  MoveL (T18849) to (113.75, 117.08, 19.7) mm, rotated rx 180 ry 0 rz -180 deg; joints [1.869, 69.168, -34.061, 3.247, -35.151, -2.656]
  Call Extruder 0.34538
  MoveL (T18850) to (108.6, 106.98, 19.7) mm, rotated rx 180 ry 0 rz -180 deg; joints [1.874, 68.733, -33.242, 3.226, -35.533, -2.626]
  Call Extruder 0.01947
  MoveL (T18851) to (108.6, 106.34, 19.7) mm, rotated rx 180 ry 0 rz -180 deg; joints [1.874, 68.733, -33.242, 3.226, -35.533, -2.626]
  Set speed (150.0 mm/s)
  MoveL (T18852) to (108.54, 105.89, 19.7) mm, rotated rx 180 ry 0 rz -180 deg; joints [1.874, 68.733, -33.242, 3.226, -35.533, -2.626]
  Set speed (45.0 mm/s)
  Call Extruder -1.6
  MoveL (T18853) to (108.54, 105.89, 19.7) mm, rotated rx 180 ry 0 rz -180 deg; joints [1.866, 68.675, -33.134, 3.208, -35.583, -2.61]
  Set speed (120.0 mm/s)
  MoveL (T18854) to (108.54, 105.89, 19.7) mm, rotated rx 180 ry 0 rz -180 deg; joints [1.866, 68.675, -33.134, 3.208, -35.583, -2.61]
  Call Extruder -0.38
  MoveL (T18855) to (109.66, 106.33, 19.7) mm, rotated rx 180 ry 0 rz -180 deg; joints [1.815, 68.53, -32.862, 3.11, -35.708, -2.526]
  Set speed (45.0 mm/s)
  Call Extruder -0.02
  MoveL (T18856) to (109.66, 106.33, 19.7) mm, rotated rx 180 ry 0 rz -180 deg; joints [1.815, 68.53, -32.862, 3.11, -35.708, -2.526]
  Set speed (150.0 mm/s)
  MoveL (T18857) to (109.66, 106.33, 21.7) mm, rotated rx 180 ry 0 rz -180 deg; joints [2.818, 66.213, -28.512, 4.602, -37.791, -3.64]
  MoveL (T18858) to (104.34, 103.54, 21.7) mm, rotated rx 180 ry 0 rz -180 deg; joints [2.818, 66.213, -28.512, 4.602, -37.791, -3.64]
  MoveL (T18859) to (104.34, 103.54, 19.7) mm, rotated rx 180 ry 0 rz -180 deg; joints [2.938, 66.228, -28.539, 4.799, -37.786, -3.796]
  Set speed (40.0 mm/s)
  Call Extruder 2.0
  MoveL (T18860) to (104.34, 103.54, 19.7) mm, rotated rx 180 ry 0 rz -180 deg; joints [2.938, 66.228, -28.539, 4.799, -37.786, -3.796]
  Call Extruder 0.52159
  MoveL (T18861) to (121.46, 103.54, 19.7) mm, rotated rx 180 ry 0 rz -180 deg; joints [2.938, 66.228, -28.539, 4.799, -37.786, -3.796]
  Call Extruder 0.54596
  MoveL (T18862) to (121.46, 121.46, 19.7) mm, rotated rx 180 ry 0 rz -180 deg; joints [2.938, 66.228, -28.539, 4.799, -37.786, -3.796]
  Call Extruder 0.54596
  MoveL (T18863) to (103.54, 121.46, 19.7) mm, rotated rx 180 ry 0 rz -180 deg; joints [3.295, 67.194, -30.352, 5.484, -36.967, -4.386]
  Call Extruder 0.54596
  MoveL (T18864) to (103.54, 103.54, 19.7) mm, rotated rx 180 ry 0 rz -180 deg; joints [3.288, 67.492, -30.912, 5.506, -36.706, -4.419]
  Call Extruder 0.02254
  MoveL (T18865) to (104.28, 103.54, 19.7) mm, rotated rx 180 ry 0 rz -180 deg; joints [3.288, 67.492, -30.912, 5.506, -36.706, -4.419]
  Set speed (150.0 mm/s)
  MoveL (T18866) to (103.53, 103.13, 19.7) mm, rotated rx 180 ry 0 rz -180 deg; joints [3.288, 67.492, -30.912, 5.506, -36.706, -4.419]
  Set speed (40.0 mm/s)
  MoveL (T18867) to (103.53, 103.13, 19.7) mm, rotated rx 180 ry 0 rz -180 deg; joints [2.356, 69.73, -35.116, 4.142, -34.684, -3.408]
  Call Extruder 0.55858
  MoveL (T18868) to (121.87, 103.13, 19.7) mm, rotated rx 180 ry 0 rz -180 deg; joints [2.356, 69.73, -35.116, 4.142, -34.684, -3.408]
  Call Extruder 0.57077
  MoveL (T18869) to (121.87, 121.87, 19.7) mm, rotated rx 180 ry 0 rz -180 deg; joints [2.29, 69.723, -35.102, 4.026, -34.687, -3.312]
  Call Extruder 0.57077
  MoveL (T18870) to (103.13, 121.87, 19.7) mm, rotated rx 180 ry 0 rz -180 deg; joints [2.29, 69.723, -35.102, 4.026, -34.687, -3.312]
  Call Extruder 0.57077
  MoveL (T18871) to (103.13, 103.13, 19.7) mm, rotated rx 180 ry 0 rz -180 deg; joints [1.775, 68.231, -32.301, 3.023, -35.968, -2.447]
  Call Extruder 0.01036
  MoveL (T18872) to (103.47, 103.13, 19.7) mm, rotated rx 180 ry 0 rz -180 deg; joints [1.775, 68.231, -32.301, 3.023, -35.968, -2.447]
  Set speed (150.0 mm/s)
  MoveL (T18873) to (102.72, 102.81, 19.7) mm, rotated rx 180 ry 0 rz -180 deg; joints [1.875, 67.989, -31.846, 3.176, -36.185, -2.565]
  Set speed (25.0 mm/s)
  MoveL (T18874) to (102.72, 102.81, 19.7) mm, rotated rx 180 ry 0 rz -180 deg; joints [1.875, 67.989, -31.846, 3.176, -36.185, -2.565]
  Call Extruder 0.00259
  MoveL (T18875) to (102.72, 102.72, 19.7) mm, rotated rx 180 ry 0 rz -180 deg; joints [1.875, 67.989, -31.846, 3.176, -36.185, -2.565]
  Call Extruder 0.59557
  MoveL (T18876) to (122.28, 102.72, 19.7) mm, rotated rx 180 ry 0 rz -180 deg; joints [1.875, 67.989, -31.846, 3.176, -36.185, -2.565]
  Call Extruder 0.59557
  MoveL (T18877) to (122.28, 122.28, 19.7) mm, rotated rx 180 ry 0 rz -180 deg; joints [1.884, 67.935, -31.744, 3.189, -36.233, -2.573]
  Call Extruder 0.59557
  MoveL (T18878) to (102.72, 122.28, 19.7) mm, rotated rx 180 ry 0 rz -180 deg; joints [1.888, 67.676, -31.258, 3.177, -36.46, -2.556]
  Call Extruder 0.59115
  MoveL (T18879) to (102.72, 102.87, 19.7) mm, rotated rx 180 ry 0 rz -180 deg; joints [1.888, 67.676, -31.258, 3.177, -36.46, -2.556]
  Set speed (150.0 mm/s)
  MoveL (T18880) to (102.78, 102.75, 19.7) mm, rotated rx 180 ry 0 rz -180 deg; joints [1.888, 67.676, -31.258, 3.177, -36.46, -2.556]
  Set speed (45.0 mm/s)
  Call Extruder -1.6
  MoveL (T18881) to (102.78, 102.75, 19.7) mm, rotated rx 180 ry 0 rz -180 deg; joints [1.888, 67.676, -31.258, 3.177, -36.46, -2.556]
  Set speed (120.0 mm/s)
  MoveL (T18882) to (102.78, 102.75, 19.7) mm, rotated rx 180 ry 0 rz -180 deg; joints [1.888, 67.676, -31.258, 3.177, -36.46, -2.556]
  Call Extruder -0.05166
  MoveL (T18883) to (102.72, 102.72, 19.7) mm, rotated rx 180 ry 0 rz -180 deg; joints [1.888, 67.676, -31.258, 3.177, -36.46, -2.556]
  Call Extruder -0.32834
  MoveL (T18884) to (103.65, 102.72, 19.7) mm, rotated rx 180 ry 0 rz -180 deg; joints [1.888, 67.676, -31.258, 3.177, -36.46, -2.556]
  Set speed (45.0 mm/s)
  Call Extruder -0.02
  MoveL (T18885) to (103.65, 102.72, 19.7) mm, rotated rx 180 ry 0 rz -180 deg; joints [1.888, 67.676, -31.258, 3.177, -36.46, -2.556]
  Set speed (150.0 mm/s)
  MoveL (T18886) to (103.65, 102.72, 21.7) mm, rotated rx 180 ry 0 rz -180 deg; joints [1.888, 67.676, -31.258, 3.177, -36.46, -2.556]
  MoveL (T18887) to (121.34, 120.51, 21.7) mm, rotated rx 180 ry 0 rz -180 deg; joints [1.884, 67.935, -31.744, 3.189, -36.233, -2.573]
  MoveL (T18888) to (121.34, 120.51, 19.7) mm, rotated rx 180 ry 0 rz -180 deg; joints [1.884, 67.935, -31.744, 3.189, -36.233, -2.573]
  Set speed (40.0 mm/s)
  Call Extruder 2.0
  MoveL (T18889) to (121.34, 120.51, 19.7) mm, rotated rx 180 ry 0 rz -180 deg; joints [1.884, 67.935, -31.744, 3.189, -36.233, -2.573]
  Call Extruder 0.02815
  MoveL (T18890) to (120.69, 121.16, 19.7) mm, rotated rx 180 ry 0 rz -180 deg; joints [1.879, 67.965, -31.801, 3.182, -36.206, -2.568]
  Call Extruder 0.01786
  MoveL (T18891) to (120.11, 121.16, 19.7) mm, rotated rx 180 ry 0 rz -180 deg; joints [1.879, 67.965, -31.801, 3.182, -36.206, -2.568]
  Call Extruder 0.04544
  MoveL (T18892) to (121.16, 120.11, 19.7) mm, rotated rx 180 ry 0 rz -180 deg; joints [1.879, 67.965, -31.801, 3.182, -36.206, -2.568]
  Call Extruder 0.01786
  MoveL (T18893) to (121.16, 119.53, 19.7) mm, rotated rx 180 ry 0 rz -180 deg; joints [1.879, 67.965, -31.801, 3.182, -36.206, -2.568]
  Call Extruder 0.0707
  MoveL (T18894) to (119.53, 121.16, 19.7) mm, rotated rx 180 ry 0 rz -180 deg; joints [1.879, 67.965, -31.801, 3.182, -36.206, -2.568]
  Call Extruder 0.01786
  MoveL (T18895) to (118.95, 121.16, 19.7) mm, rotated rx 180 ry 0 rz -180 deg; joints [1.879, 67.731, -31.763, 3.197, -36.01, -2.587]
  Call Extruder 0.09595
  MoveL (T18896) to (121.16, 118.95, 19.7) mm, rotated rx 180 ry 0 rz -180 deg; joints [1.476, 70.466, -36.894, 2.667, -33.601, -2.222]
  Call Extruder 0.01786
  MoveL (T18897) to (121.16, 118.37, 19.7) mm, rotated rx 180 ry 0 rz -180 deg; joints [1.476, 70.698, -36.935, 2.654, -33.792, -2.206]
  Call Extruder 0.12121
  MoveL (T18898) to (118.37, 121.16, 19.7) mm, rotated rx 180 ry 0 rz -180 deg; joints [1.476, 70.698, -36.935, 2.654, -33.792, -2.206]
  Call Extruder 0.01786
  MoveL (T18899) to (117.79, 121.16, 19.7) mm, rotated rx 180 ry 0 rz -180 deg; joints [1.476, 70.698, -36.935, 2.654, -33.792, -2.206]
  Call Extruder 0.14646
  MoveL (T18900) to (121.16, 117.79, 19.7) mm, rotated rx 180 ry 0 rz -180 deg; joints [1.476, 70.698, -36.935, 2.654, -33.792, -2.206]
  Call Extruder 0.01786
  MoveL (T18901) to (121.16, 117.21, 19.7) mm, rotated rx 180 ry 0 rz -180 deg; joints [1.476, 70.698, -36.935, 2.654, -33.792, -2.206]
  Call Extruder 0.17172
  MoveL (T18902) to (117.21, 121.16, 19.7) mm, rotated rx 180 ry 0 rz -180 deg; joints [1.476, 70.698, -36.935, 2.654, -33.792, -2.206]
  Call Extruder 0.01786
  MoveL (T18903) to (116.62, 121.16, 19.7) mm, rotated rx 180 ry 0 rz -180 deg; joints [1.476, 70.698, -36.935, 2.654, -33.792, -2.206]
  Call Extruder 0.19697
  MoveL (T18904) to (121.16, 116.62, 19.7) mm, rotated rx 180 ry 0 rz -180 deg; joints [1.476, 70.698, -36.935, 2.654, -33.792, -2.206]
  Call Extruder 0.01786
  MoveL (T18905) to (121.16, 116.04, 19.7) mm, rotated rx 180 ry 0 rz -180 deg; joints [1.4, 70.466, -36.499, 2.505, -33.993, -2.077]
  Call Extruder 0.1471
  MoveL (T18906) to (117.77, 119.43, 19.7) mm, rotated rx 180 ry 0 rz -180 deg; joints [1.402, 70.285, -36.159, 2.497, -34.152, -2.067]
  Call Extruder 0.01786
  MoveL (T18907) to (117.77, 118.85, 19.7) mm, rotated rx 180 ry 0 rz -180 deg; joints [1.402, 70.285, -36.159, 2.497, -34.152, -2.067]
  Call Extruder 0.1471
  MoveL (T18908) to (121.16, 115.46, 19.7) mm, rotated rx 180 ry 0 rz -180 deg; joints [1.402, 70.285, -36.159, 2.497, -34.152, -2.067]
  Call Extruder 0.01786
  MoveL (T18909) to (121.16, 114.88, 19.7) mm, rotated rx 180 ry 0 rz -180 deg; joints [1.402, 70.285, -36.159, 2.497, -34.152, -2.067]
  Call Extruder 0.1471
  MoveL (T18910) to (117.77, 118.27, 19.7) mm, rotated rx 180 ry 0 rz -180 deg; joints [1.52, 70.645, -36.835, 2.729, -33.84, -2.268]
  Call Extruder 0.0059
  MoveL (T18911) to (117.77, 118.07, 19.7) mm, rotated rx 180 ry 0 rz -180 deg; joints [1.582, 70.65, -36.844, 2.842, -33.839, -2.361]
  Call Extruder 0.00889
  MoveL (T18912) to (117.64, 117.82, 19.7) mm, rotated rx 180 ry 0 rz -180 deg; joints [1.582, 70.65, -36.844, 2.842, -33.839, -2.361]
  Call Extruder 0.15283
  MoveL (T18913) to (121.16, 114.3, 19.7) mm, rotated rx 180 ry 0 rz -180 deg; joints [1.582, 70.65, -36.844, 2.842, -33.839, -2.361]
  Call Extruder 0.01786
  MoveL (T18914) to (121.16, 113.72, 19.7) mm, rotated rx 180 ry 0 rz -180 deg; joints [1.403, 70.106, -35.823, 2.49, -34.309, -2.057]
  Call Extruder 0.16138
  MoveL (T18915) to (117.44, 117.43, 19.7) mm, rotated rx 180 ry 0 rz -180 deg; joints [1.403, 70.106, -35.823, 2.49, -34.309, -2.057]
  Call Extruder 0.01327
  MoveL (T18916) to (117.25, 117.05, 19.7) mm, rotated rx 180 ry 0 rz -180 deg; joints [1.403, 70.106, -35.823, 2.49, -34.309, -2.057]
  Call Extruder 0.16993
  MoveL (T18917) to (121.16, 113.14, 19.7) mm, rotated rx 180 ry 0 rz -180 deg; joints [1.405, 69.928, -35.489, 2.483, -34.465, -2.047]
  Call Extruder 0.01786
  MoveL (T18918) to (121.16, 112.56, 19.7) mm, rotated rx 180 ry 0 rz -180 deg; joints [1.405, 69.928, -35.489, 2.483, -34.465, -2.047]
  Call Extruder 0.17848
  MoveL (T18919) to (117.05, 116.66, 19.7) mm, rotated rx 180 ry 0 rz -180 deg; joints [1.405, 69.928, -35.489, 2.483, -34.465, -2.047]
  Call Extruder 0.01327
  MoveL (T18920) to (116.85, 116.28, 19.7) mm, rotated rx 180 ry 0 rz -180 deg; joints [1.405, 69.928, -35.489, 2.483, -34.465, -2.047]
  Call Extruder 0.18703
  MoveL (T18921) to (121.16, 111.98, 19.7) mm, rotated rx 180 ry 0 rz -180 deg; joints [1.656, 70.504, -36.569, 2.965, -33.97, -2.459]
  Call Extruder 0.01786
  MoveL (T18922) to (121.16, 111.4, 19.7) mm, rotated rx 180 ry 0 rz -180 deg; joints [1.656, 70.504, -36.569, 2.965, -33.97, -2.459]
  Call Extruder 0.19558
  MoveL (T18923) to (116.66, 115.89, 19.7) mm, rotated rx 180 ry 0 rz -180 deg; joints [1.406, 69.752, -35.158, 2.476, -34.62, -2.038]
  Call Extruder 0.01327
  MoveL (T18924) to (116.46, 115.51, 19.7) mm, rotated rx 180 ry 0 rz -180 deg; joints [1.406, 69.752, -35.158, 2.476, -34.62, -2.038]
  Call Extruder 0.20412
  MoveL (T18925) to (121.16, 110.81, 19.7) mm, rotated rx 180 ry 0 rz -180 deg; joints [1.408, 69.577, -34.828, 2.469, -34.773, -2.028]
  Call Extruder 0.01786
  MoveL (T18926) to (121.16, 110.23, 19.7) mm, rotated rx 180 ry 0 rz -180 deg; joints [1.408, 69.577, -34.828, 2.469, -34.773, -2.028]
  Call Extruder 0.21267
  MoveL (T18927) to (116.26, 115.13, 19.7) mm, rotated rx 180 ry 0 rz -180 deg; joints [1.688, 70.415, -36.404, 3.016, -34.049, -2.5]
  Call Extruder 0.01327
  MoveL (T18928) to (116.07, 114.74, 19.7) mm, rotated rx 180 ry 0 rz -180 deg; joints [1.688, 70.415, -36.404, 3.016, -34.049, -2.5]
  Call Extruder 0.22122
  MoveL (T18929) to (121.16, 109.65, 19.7) mm, rotated rx 180 ry 0 rz -180 deg; joints [1.688, 70.415, -36.404, 3.016, -34.049, -2.5]
  Call Extruder 0.01786
  MoveL (T18930) to (121.16, 109.07, 19.7) mm, rotated rx 180 ry 0 rz -180 deg; joints [1.72, 70.328, -36.239, 3.067, -34.127, -2.54]
  Call Extruder 0.22977
  MoveL (T18931) to (115.87, 114.36, 19.7) mm, rotated rx 180 ry 0 rz -180 deg; joints [1.72, 70.328, -36.239, 3.067, -34.127, -2.54]
  Call Extruder 0.01327
  MoveL (T18932) to (115.67, 113.97, 19.7) mm, rotated rx 180 ry 0 rz -180 deg; joints [1.72, 70.328, -36.239, 3.067, -34.127, -2.54]
  Call Extruder 0.23832
  MoveL (T18933) to (121.16, 108.49, 19.7) mm, rotated rx 180 ry 0 rz -180 deg; joints [1.409, 69.403, -34.502, 2.462, -34.926, -2.019]
  Call Extruder 0.01786
  MoveL (T18934) to (121.16, 107.91, 19.7) mm, rotated rx 180 ry 0 rz -180 deg; joints [1.409, 69.403, -34.502, 2.462, -34.926, -2.019]
  Call Extruder 0.24687
  MoveL (T18935) to (115.48, 113.59, 19.7) mm, rotated rx 180 ry 0 rz -180 deg; joints [1.411, 69.231, -34.178, 2.456, -35.077, -2.01]
  Call Extruder 0.01327
  MoveL (T18936) to (115.28, 113.2, 19.7) mm, rotated rx 180 ry 0 rz -180 deg; joints [1.411, 69.231, -34.178, 2.456, -35.077, -2.01]
  Call Extruder 0.25542
  MoveL (T18937) to (121.16, 107.33, 19.7) mm, rotated rx 180 ry 0 rz -180 deg; joints [1.411, 69.231, -34.178, 2.456, -35.077, -2.01]
  Call Extruder 0.01786
  MoveL (T18938) to (121.16, 106.75, 19.7) mm, rotated rx 180 ry 0 rz -180 deg; joints [1.753, 70.241, -36.076, 3.119, -34.205, -2.58]
  Call Extruder 0.26397
  MoveL (T18939) to (115.08, 112.82, 19.7) mm, rotated rx 180 ry 0 rz -180 deg; joints [1.753, 70.241, -36.076, 3.119, -34.205, -2.58]
  Call Extruder 0.01327
  MoveL (T18940) to (114.89, 112.44, 19.7) mm, rotated rx 180 ry 0 rz -180 deg; joints [1.753, 70.241, -36.076, 3.119, -34.205, -2.58]
  Call Extruder 0.27252
  MoveL (T18941) to (121.16, 106.17, 19.7) mm, rotated rx 180 ry 0 rz -180 deg; joints [1.785, 70.154, -35.913, 3.17, -34.282, -2.62]
  Call Extruder 0.01786
  MoveL (T18942) to (121.16, 105.59, 19.7) mm, rotated rx 180 ry 0 rz -180 deg; joints [1.785, 70.154, -35.913, 3.17, -34.282, -2.62]
  Call Extruder 0.13907
  MoveL (T18943) to (117.96, 108.79, 19.7) mm, rotated rx 180 ry 0 rz -180 deg; joints [1.785, 70.154, -35.913, 3.17, -34.282, -2.62]
  Call Extruder 0.01777
  MoveL (T18944) to (117.96, 109.36, 19.7) mm, rotated rx 180 ry 0 rz -180 deg; joints [1.412, 69.059, -33.856, 2.449, -35.228, -2.001]
  Call Extruder 0.01777
  MoveL (T18945) to (117.38, 109.36, 19.7) mm, rotated rx 180 ry 0 rz -180 deg; joints [1.412, 69.059, -33.856, 2.449, -35.228, -2.001]
  Call Extruder 0.11687
  MoveL (T18946) to (114.69, 112.05, 19.7) mm, rotated rx 180 ry 0 rz -180 deg; joints [1.414, 68.89, -33.537, 2.443, -35.377, -1.992]
  Call Extruder 0.01327
  MoveL (T18947) to (114.49, 111.67, 19.7) mm, rotated rx 180 ry 0 rz -180 deg; joints [1.414, 68.89, -33.537, 2.443, -35.377, -1.992]
  Call Extruder 0.10016
  MoveL (T18948) to (116.8, 109.36, 19.7) mm, rotated rx 180 ry 0 rz -180 deg; joints [1.815, 70.063, -35.741, 3.217, -34.364, -2.657]
  Call Extruder 0.01786
  MoveL (T18949) to (116.22, 109.36, 19.7) mm, rotated rx 180 ry 0 rz -180 deg; joints [1.815, 70.063, -35.741, 3.217, -34.364, -2.657]
  Call Extruder 0.08346
  MoveL (T18950) to (114.3, 111.28, 19.7) mm, rotated rx 180 ry 0 rz -180 deg; joints [1.817, 69.885, -35.407, 3.208, -34.52, -2.644]
  Call Extruder 0.01327
  MoveL (T18951) to (114.1, 110.9, 19.7) mm, rotated rx 180 ry 0 rz -180 deg; joints [1.817, 69.885, -35.407, 3.208, -34.52, -2.644]
  Call Extruder 0.06675
  MoveL (T18952) to (115.64, 109.36, 19.7) mm, rotated rx 180 ry 0 rz -180 deg; joints [1.416, 68.72, -33.22, 2.437, -35.525, -1.983]
  Call Extruder 0.01786
  MoveL (T18953) to (115.06, 109.36, 19.7) mm, rotated rx 180 ry 0 rz -180 deg; joints [1.416, 68.72, -33.22, 2.437, -35.525, -1.983]
  Call Extruder 0.05004
  MoveL (T18954) to (113.9, 110.52, 19.7) mm, rotated rx 180 ry 0 rz -180 deg; joints [1.416, 68.72, -33.22, 2.437, -35.525, -1.983]
  Call Extruder 0.01327
  MoveL (T18955) to (113.71, 110.13, 19.7) mm, rotated rx 180 ry 0 rz -180 deg; joints [1.417, 68.553, -32.905, 2.431, -35.672, -1.975]
  Call Extruder 0.03334
  MoveL (T18956) to (114.47, 109.36, 19.7) mm, rotated rx 180 ry 0 rz -180 deg; joints [1.417, 68.553, -32.905, 2.431, -35.672, -1.975]
  Call Extruder 0.01786
  MoveL (T18957) to (113.89, 109.36, 19.7) mm, rotated rx 180 ry 0 rz -180 deg; joints [1.417, 68.553, -32.905, 2.431, -35.672, -1.975]
  Call Extruder 0.02255
  MoveL (T18958) to (113.37, 109.88, 19.7) mm, rotated rx 180 ry 0 rz -180 deg; joints [1.819, 69.709, -35.077, 3.199, -34.674, -2.632]
  Set speed (45.0 mm/s)
  Call Extruder -1.6
  MoveL (T18959) to (113.37, 109.88, 19.7) mm, rotated rx 180 ry 0 rz -180 deg; joints [1.819, 69.709, -35.077, 3.199, -34.674, -2.632]
  Set speed (120.0 mm/s)
  MoveL (T18960) to (113.37, 109.88, 19.7) mm, rotated rx 180 ry 0 rz -180 deg; joints [1.819, 69.709, -35.077, 3.199, -34.674, -2.632]
  Call Extruder -0.26134
  MoveL (T18961) to (113.89, 109.36, 19.7) mm, rotated rx 180 ry 0 rz -180 deg; joints [1.821, 69.535, -34.749, 3.19, -34.827, -2.62]
  Call Extruder -0.11866
  MoveL (T18962) to (114.23, 109.36, 19.7) mm, rotated rx 180 ry 0 rz -180 deg; joints [1.821, 69.535, -34.749, 3.19, -34.827, -2.62]
  Set speed (45.0 mm/s)
  Call Extruder -0.02
  MoveL (T18963) to (114.23, 109.36, 19.7) mm, rotated rx 180 ry 0 rz -180 deg; joints [1.419, 68.386, -32.592, 2.425, -35.819, -1.966]
  Set speed (150.0 mm/s)
  MoveL (T18964) to (114.23, 109.36, 21.7) mm, rotated rx 180 ry 0 rz -180 deg; joints [1.419, 68.386, -32.592, 2.425, -35.819, -1.966]
  MoveL (T18965) to (117.77, 108.39, 21.7) mm, rotated rx 180 ry 0 rz -180 deg; joints [1.419, 68.386, -32.592, 2.425, -35.819, -1.966]
  MoveL (T18966) to (117.77, 108.39, 19.7) mm, rotated rx 180 ry 0 rz -180 deg; joints [1.42, 68.221, -32.281, 2.419, -35.964, -1.958]
  Set speed (40.0 mm/s)
  Call Extruder 2.0
  MoveL (T18967) to (117.77, 108.39, 19.7) mm, rotated rx 180 ry 0 rz -180 deg; joints [1.42, 68.221, -32.281, 2.419, -35.964, -1.958]
  Call Extruder 0.14703
  MoveL (T18968) to (121.16, 105.01, 19.7) mm, rotated rx 180 ry 0 rz -180 deg; joints [1.823, 69.361, -34.423, 3.182, -34.98, -2.608]
  Call Extruder 0.01786
  MoveL (T18969) to (121.16, 104.42, 19.7) mm, rotated rx 180 ry 0 rz -180 deg; joints [1.823, 69.361, -34.423, 3.182, -34.98, -2.608]
  Call Extruder 0.13907
  MoveL (T18970) to (117.96, 107.62, 19.7) mm, rotated rx 180 ry 0 rz -180 deg; joints [1.823, 69.361, -34.423, 3.182, -34.98, -2.608]
  Call Extruder 0.01786
  MoveL (T18971) to (117.96, 107.04, 19.7) mm, rotated rx 180 ry 0 rz -180 deg; joints [1.825, 69.189, -34.1, 3.173, -35.131, -2.596]
  Call Extruder 0.13906
  MoveL (T18972) to (121.16, 103.84, 19.7) mm, rotated rx 180 ry 0 rz -180 deg; joints [1.825, 69.189, -34.1, 3.173, -35.131, -2.596]
  Call Extruder 0.01786
  MoveL (T18973) to (120.58, 103.84, 19.7) mm, rotated rx 180 ry 0 rz -180 deg; joints [1.422, 68.056, -31.973, 2.413, -36.108, -1.95]
  Call Extruder 0.11381
  MoveL (T18974) to (117.96, 106.46, 19.7) mm, rotated rx 180 ry 0 rz -180 deg; joints [1.422, 68.056, -31.973, 2.413, -36.108, -1.95]
  Call Extruder 0.01786
  MoveL (T18975) to (117.96, 105.88, 19.7) mm, rotated rx 180 ry 0 rz -180 deg; joints [1.422, 68.056, -31.973, 2.413, -36.108, -1.95]
  Call Extruder 0.08856
  MoveL (T18976) to (119.99, 103.84, 19.7) mm, rotated rx 180 ry 0 rz -180 deg; joints [1.423, 67.893, -31.665, 2.408, -36.252, -1.942]
  Call Extruder 0.01786
  MoveL (T18977) to (119.41, 103.84, 19.7) mm, rotated rx 180 ry 0 rz -180 deg; joints [1.423, 67.893, -31.665, 2.408, -36.252, -1.942]
  Call Extruder 0.0633
  MoveL (T18978) to (117.96, 105.3, 19.7) mm, rotated rx 180 ry 0 rz -180 deg; joints [1.827, 69.018, -33.778, 3.165, -35.281, -2.585]
  Call Extruder 0.00424
  MoveL (T18979) to (117.96, 105.16, 19.7) mm, rotated rx 180 ry 0 rz -180 deg; joints [1.827, 69.018, -33.778, 3.165, -35.281, -2.585]
  Call Extruder 0.01362
  MoveL (T18980) to (117.51, 105.16, 19.7) mm, rotated rx 180 ry 0 rz -180 deg; joints [1.827, 69.018, -33.778, 3.165, -35.281, -2.585]
  Call Extruder 0.0573
  MoveL (T18981) to (118.83, 103.84, 19.7) mm, rotated rx 180 ry 0 rz -180 deg; joints [1.829, 68.848, -33.46, 3.157, -35.43, -2.573]
  Call Extruder 0.01786
  MoveL (T18982) to (118.25, 103.84, 19.7) mm, rotated rx 180 ry 0 rz -180 deg; joints [1.829, 68.848, -33.46, 3.157, -35.43, -2.573]
  Call Extruder 0.0573
  MoveL (T18983) to (116.93, 105.16, 19.7) mm, rotated rx 180 ry 0 rz -180 deg; joints [1.829, 68.848, -33.46, 3.157, -35.43, -2.573]
  Call Extruder 0.01786
  MoveL (T18984) to (116.35, 105.16, 19.7) mm, rotated rx 180 ry 0 rz -180 deg; joints [1.425, 67.731, -31.361, 2.402, -36.394, -1.934]
  Call Extruder 0.0573
  MoveL (T18985) to (117.67, 103.84, 19.7) mm, rotated rx 180 ry 0 rz -180 deg; joints [1.425, 67.731, -31.361, 2.402, -36.394, -1.934]
  Call Extruder 0.01786
  MoveL (T18986) to (117.09, 103.84, 19.7) mm, rotated rx 180 ry 0 rz -180 deg; joints [1.425, 67.731, -31.361, 2.402, -36.394, -1.934]
  Call Extruder 0.0573
  MoveL (T18987) to (115.77, 105.16, 19.7) mm, rotated rx 180 ry 0 rz -180 deg; joints [1.427, 67.569, -31.058, 2.397, -36.535, -1.926]
  Call Extruder 0.01786
  MoveL (T18988) to (115.19, 105.16, 19.7) mm, rotated rx 180 ry 0 rz -180 deg; joints [1.427, 67.569, -31.058, 2.397, -36.535, -1.926]
  Call Extruder 0.0573
  MoveL (T18989) to (116.51, 103.84, 19.7) mm, rotated rx 180 ry 0 rz -180 deg; joints [1.69, 68.284, -32.4, 2.882, -35.919, -2.335]
  Call Extruder 0.01786
  MoveL (T18990) to (115.93, 103.84, 19.7) mm, rotated rx 180 ry 0 rz -180 deg; joints [1.69, 68.284, -32.4, 2.882, -35.919, -2.335]
  Call Extruder 0.0573
  MoveL (T18991) to (114.61, 105.16, 19.7) mm, rotated rx 180 ry 0 rz -180 deg; joints [1.723, 68.204, -32.249, 2.932, -35.99, -2.373]
  Call Extruder 0.01786
  MoveL (T18992) to (114.03, 105.16, 19.7) mm, rotated rx 180 ry 0 rz -180 deg; joints [1.723, 68.204, -32.249, 2.932, -35.99, -2.373]
  Call Extruder 0.0573
  MoveL (T18993) to (115.35, 103.84, 19.7) mm, rotated rx 180 ry 0 rz -180 deg; joints [1.723, 68.204, -32.249, 2.932, -35.99, -2.373]
  Call Extruder 0.01786
  MoveL (T18994) to (114.77, 103.84, 19.7) mm, rotated rx 180 ry 0 rz -180 deg; joints [1.428, 67.409, -30.757, 2.391, -36.676, -1.918]
  Call Extruder 0.0573
  MoveL (T18995) to (113.45, 105.16, 19.7) mm, rotated rx 180 ry 0 rz -180 deg; joints [1.428, 67.409, -30.757, 2.391, -36.676, -1.918]
  Call Extruder 0.01786
  MoveL (T18996) to (112.87, 105.16, 19.7) mm, rotated rx 180 ry 0 rz -180 deg; joints [1.428, 67.409, -30.757, 2.391, -36.676, -1.918]
  Call Extruder 0.0573
  MoveL (T18997) to (114.18, 103.84, 19.7) mm, rotated rx 180 ry 0 rz -180 deg; joints [1.43, 67.249, -30.457, 2.386, -36.816, -1.911]
  Call Extruder 0.01786
  MoveL (T18998) to (113.6, 103.84, 19.7) mm, rotated rx 180 ry 0 rz -180 deg; joints [1.43, 67.249, -30.457, 2.386, -36.816, -1.911]
  Call Extruder 0.0573
  MoveL (T18999) to (112.28, 105.16, 19.7) mm, rotated rx 180 ry 0 rz -180 deg; joints [1.755, 68.124, -32.099, 2.983, -36.062, -2.412]
  Call Extruder 0.01786
  MoveL (T19000) to (111.7, 105.16, 19.7) mm, rotated rx 180 ry 0 rz -180 deg; joints [1.788, 68.044, -31.95, 3.033, -36.133, -2.451]
  Call Extruder 0.0573
  MoveL (T19001) to (113.02, 103.84, 19.7) mm, rotated rx 180 ry 0 rz -180 deg; joints [1.788, 68.044, -31.95, 3.033, -36.133, -2.451]
  Call Extruder 0.01786
  MoveL (T19002) to (112.44, 103.84, 19.7) mm, rotated rx 180 ry 0 rz -180 deg; joints [1.431, 67.091, -30.16, 2.381, -36.955, -1.903]
  Call Extruder 0.0573
  MoveL (T19003) to (111.12, 105.16, 19.7) mm, rotated rx 180 ry 0 rz -180 deg; joints [1.431, 67.091, -30.16, 2.381, -36.955, -1.903]
  Call Extruder 0.01786
  MoveL (T19004) to (110.54, 105.16, 19.7) mm, rotated rx 180 ry 0 rz -180 deg; joints [1.431, 67.091, -30.16, 2.381, -36.955, -1.903]
  Call Extruder 0.0573
  MoveL (T19005) to (111.86, 103.84, 19.7) mm, rotated rx 180 ry 0 rz -180 deg; joints [1.433, 66.934, -29.865, 2.376, -37.093, -1.896]
  Call Extruder 0.01786
  MoveL (T19006) to (111.28, 103.84, 19.7) mm, rotated rx 180 ry 0 rz -180 deg; joints [1.433, 66.934, -29.865, 2.376, -37.093, -1.896]
  Call Extruder 0.0573
  MoveL (T19007) to (109.96, 105.16, 19.7) mm, rotated rx 180 ry 0 rz -180 deg; joints [1.433, 66.934, -29.865, 2.376, -37.093, -1.896]
  Call Extruder 0.01786
  MoveL (T19008) to (109.38, 105.16, 19.7) mm, rotated rx 180 ry 0 rz -180 deg; joints [1.821, 67.965, -31.801, 3.084, -36.203, -2.489]
  Call Extruder 0.0573
  MoveL (T19009) to (110.7, 103.84, 19.7) mm, rotated rx 180 ry 0 rz -180 deg; joints [1.821, 67.965, -31.801, 3.084, -36.203, -2.489]
  Call Extruder 0.01786
  MoveL (T19010) to (110.12, 103.84, 19.7) mm, rotated rx 180 ry 0 rz -180 deg; joints [1.821, 67.965, -31.801, 3.084, -36.203, -2.489]
  Call Extruder 0.0573
  MoveL (T19011) to (108.8, 105.16, 19.7) mm, rotated rx 180 ry 0 rz -180 deg; joints [1.838, 67.923, -31.721, 3.111, -36.242, -2.51]
  Call Extruder 0.01786
  MoveL (T19012) to (108.22, 105.16, 19.7) mm, rotated rx 180 ry 0 rz -180 deg; joints [1.838, 67.923, -31.721, 3.111, -36.242, -2.51]
  Call Extruder 0.06527
  MoveL (T19013) to (109.72, 103.66, 19.7) mm, rotated rx 180 ry 0 rz -180 deg; joints [1.838, 67.923, -31.721, 3.111, -36.242, -2.51]
  Set speed (45.0 mm/s)
  Call Extruder -1.6
  MoveL (T19014) to (109.72, 103.66, 19.7) mm, rotated rx 180 ry 0 rz -180 deg; joints [1.841, 67.909, -31.695, 3.114, -36.254, -2.512]
  Set speed (120.0 mm/s)
  MoveL (T19015) to (109.72, 103.66, 19.7) mm, rotated rx 180 ry 0 rz -180 deg; joints [1.841, 67.909, -31.695, 3.114, -36.254, -2.512]
  Call Extruder -0.38
  MoveL (T19016) to (108.97, 104.42, 19.7) mm, rotated rx 180 ry 0 rz -180 deg; joints [1.842, 67.853, -31.591, 3.112, -36.302, -2.509]
  Set speed (45.0 mm/s)
  Call Extruder -0.02
  MoveL (T19017) to (108.97, 104.42, 19.7) mm, rotated rx 180 ry 0 rz -180 deg; joints [1.435, 66.777, -29.571, 2.371, -37.23, -1.889]
  Set speed (150.0 mm/s)
  MoveL (T19018) to (108.97, 104.42, 21.7) mm, rotated rx 180 ry 0 rz -180 deg; joints [1.435, 66.777, -29.571, 2.371, -37.23, -1.889]
  MoveL (T19019) to (111.87, 115.45, 21.7) mm, rotated rx 180 ry 0 rz -180 deg; joints [1.435, 66.777, -29.571, 2.371, -37.23, -1.889]
  MoveL (T19020) to (111.87, 115.45, 19.7) mm, rotated rx 180 ry 0 rz -180 deg; joints [1.435, 66.777, -29.571, 2.371, -37.23, -1.889]
  Set speed (40.0 mm/s)
  Call Extruder 2.0
  MoveL (T19021) to (111.87, 115.45, 19.7) mm, rotated rx 180 ry 0 rz -180 deg; joints [1.436, 66.621, -29.279, 2.367, -37.367, -1.881]
  Call Extruder 0.022
  MoveL (T19022) to (111.36, 115.96, 19.7) mm, rotated rx 180 ry 0 rz -180 deg; joints [1.436, 66.621, -29.279, 2.367, -37.367, -1.881]
  Call Extruder 0.01786
  MoveL (T19023) to (110.78, 115.96, 19.7) mm, rotated rx 180 ry 0 rz -180 deg; joints [1.844, 67.691, -31.287, 3.105, -36.444, -2.498]
  Call Extruder 0.03281
  MoveL (T19024) to (111.54, 115.21, 19.7) mm, rotated rx 180 ry 0 rz -180 deg; joints [1.844, 67.691, -31.287, 3.105, -36.444, -2.498]
  Call Extruder 0.01328
  MoveL (T19025) to (111.34, 114.82, 19.7) mm, rotated rx 180 ry 0 rz -180 deg; joints [1.844, 67.691, -31.287, 3.105, -36.444, -2.498]
  Call Extruder 0.04953
  MoveL (T19026) to (110.2, 115.96, 19.7) mm, rotated rx 180 ry 0 rz -180 deg; joints [1.846, 67.53, -30.985, 3.098, -36.586, -2.488]
  Call Extruder 0.01786
  MoveL (T19027) to (109.62, 115.96, 19.7) mm, rotated rx 180 ry 0 rz -180 deg; joints [1.846, 67.53, -30.985, 3.098, -36.586, -2.488]
  Call Extruder 0.06625
  MoveL (T19028) to (111.14, 114.44, 19.7) mm, rotated rx 180 ry 0 rz -180 deg; joints [1.846, 67.53, -30.985, 3.098, -36.586, -2.488]
  Call Extruder 0.01328
  MoveL (T19029) to (110.95, 114.05, 19.7) mm, rotated rx 180 ry 0 rz -180 deg; joints [1.846, 67.53, -30.985, 3.098, -36.586, -2.488]
  Call Extruder 0.08298
  MoveL (T19030) to (109.04, 115.96, 19.7) mm, rotated rx 180 ry 0 rz -180 deg; joints [1.438, 66.467, -28.988, 2.362, -37.502, -1.874]
  Call Extruder 0.01786
  MoveL (T19031) to (108.46, 115.96, 19.7) mm, rotated rx 180 ry 0 rz -180 deg; joints [1.438, 66.467, -28.988, 2.362, -37.502, -1.874]
  Call Extruder 0.10562
  MoveL (T19032) to (110.89, 113.53, 19.7) mm, rotated rx 180 ry 0 rz -180 deg; joints [1.438, 66.467, -28.988, 2.362, -37.502, -1.874]
  Set speed (45.0 mm/s)
  Call Extruder -1.6
  MoveL (T19033) to (110.89, 113.53, 19.7) mm, rotated rx 180 ry 0 rz -180 deg; joints [1.439, 66.313, -28.699, 2.357, -37.637, -1.867]
  Set speed (120.0 mm/s)
  MoveL (T19034) to (110.89, 113.53, 19.7) mm, rotated rx 180 ry 0 rz -180 deg; joints [1.439, 66.313, -28.699, 2.357, -37.637, -1.867]
  Call Extruder -0.38
  MoveL (T19035) to (110.13, 114.29, 19.7) mm, rotated rx 180 ry 0 rz -180 deg; joints [1.439, 66.313, -28.699, 2.357, -37.637, -1.867]
  Set speed (45.0 mm/s)
  Call Extruder -0.02
  MoveL (T19036) to (110.13, 114.29, 19.7) mm, rotated rx 180 ry 0 rz -180 deg; joints [1.848, 67.37, -30.684, 3.091, -36.726, -2.478]
  Set speed (150.0 mm/s)
  MoveL (T19037) to (110.13, 114.29, 21.7) mm, rotated rx 180 ry 0 rz -180 deg; joints [1.848, 67.37, -30.684, 3.091, -36.726, -2.478]
  MoveL (T19038) to (117.22, 119.98, 21.7) mm, rotated rx 180 ry 0 rz -180 deg; joints [1.85, 67.211, -30.386, 3.084, -36.865, -2.468]
  MoveL (T19039) to (117.22, 119.98, 19.7) mm, rotated rx 180 ry 0 rz -180 deg; joints [1.85, 67.211, -30.386, 3.084, -36.865, -2.468]
  Set speed (40.0 mm/s)
  Call Extruder 2.0
  MoveL (T19040) to (117.22, 119.98, 19.7) mm, rotated rx 180 ry 0 rz -180 deg; joints [1.85, 67.211, -30.386, 3.084, -36.865, -2.468]
  Call Extruder 0.05113
  MoveL (T19041) to (116.04, 121.16, 19.7) mm, rotated rx 180 ry 0 rz -180 deg; joints [1.85, 67.211, -30.386, 3.084, -36.865, -2.468]
  Call Extruder 0.01786
  MoveL (T19042) to (115.46, 121.16, 19.7) mm, rotated rx 180 ry 0 rz -180 deg; joints [1.85, 67.211, -30.386, 3.084, -36.865, -2.468]
  Call Extruder 0.04317
  MoveL (T19043) to (116.46, 120.16, 19.7) mm, rotated rx 180 ry 0 rz -180 deg; joints [1.456, 66.198, -28.484, 2.38, -37.738, -1.883]
  Call Extruder 0.01786
  MoveL (T19044) to (115.88, 120.16, 19.7) mm, rotated rx 180 ry 0 rz -180 deg; joints [1.456, 66.198, -28.484, 2.38, -37.738, -1.883]
  Call Extruder 0.04317
  MoveL (T19045) to (114.88, 121.16, 19.7) mm, rotated rx 180 ry 0 rz -180 deg; joints [1.456, 66.198, -28.484, 2.38, -37.738, -1.883]
  Call Extruder 0.01786
  MoveL (T19046) to (114.3, 121.16, 19.7) mm, rotated rx 180 ry 0 rz -180 deg; joints [1.521, 66.202, -28.492, 2.485, -37.737, -1.966]
  Call Extruder 0.04317
  MoveL (T19047) to (115.29, 120.16, 19.7) mm, rotated rx 180 ry 0 rz -180 deg; joints [1.521, 66.202, -28.492, 2.485, -37.737, -1.966]
  Call Extruder 0.01786
  MoveL (T19048) to (114.71, 120.16, 19.7) mm, rotated rx 180 ry 0 rz -180 deg; joints [1.852, 67.053, -30.089, 3.078, -37.004, -2.459]
  Call Extruder 0.04317
  MoveL (T19049) to (113.72, 121.16, 19.7) mm, rotated rx 180 ry 0 rz -180 deg; joints [1.852, 67.053, -30.089, 3.078, -37.004, -2.459]
  Call Extruder 0.01786
  MoveL (T19050) to (113.14, 121.16, 19.7) mm, rotated rx 180 ry 0 rz -180 deg; joints [1.854, 66.896, -29.794, 3.071, -37.142, -2.449]
  Call Extruder 0.04317
  MoveL (T19051) to (114.13, 120.16, 19.7) mm, rotated rx 180 ry 0 rz -180 deg; joints [1.854, 66.896, -29.794, 3.071, -37.142, -2.449]
  Call Extruder 0.01786
  MoveL (T19052) to (113.55, 120.16, 19.7) mm, rotated rx 180 ry 0 rz -180 deg; joints [1.585, 66.207, -28.5, 2.591, -37.735, -2.049]
  Call Extruder 0.04317
  MoveL (T19053) to (112.56, 121.16, 19.7) mm, rotated rx 180 ry 0 rz -180 deg; joints [1.585, 66.207, -28.5, 2.591, -37.735, -2.049]
  Call Extruder 0.01786
  MoveL (T19054) to (111.98, 121.16, 19.7) mm, rotated rx 180 ry 0 rz -180 deg; joints [1.647, 66.211, -28.508, 2.692, -37.734, -2.13]
  Call Extruder 0.04317
  MoveL (T19055) to (112.97, 120.16, 19.7) mm, rotated rx 180 ry 0 rz -180 deg; joints [1.647, 66.211, -28.508, 2.692, -37.734, -2.13]
  Call Extruder 0.01786
  MoveL (T19056) to (112.39, 120.16, 19.7) mm, rotated rx 180 ry 0 rz -180 deg; joints [1.647, 66.211, -28.508, 2.692, -37.734, -2.13]
  Call Extruder 0.04317
  MoveL (T19057) to (111.4, 121.16, 19.7) mm, rotated rx 180 ry 0 rz -180 deg; joints [1.651, 66.215, -28.516, 2.699, -37.73, -2.135]
  Call Extruder 0.01786
  MoveL (T19058) to (110.81, 121.16, 19.7) mm, rotated rx 180 ry 0 rz -180 deg; joints [1.651, 66.215, -28.516, 2.699, -37.73, -2.135]
  Call Extruder 0.04317
  MoveL (T19059) to (111.81, 120.16, 19.7) mm, rotated rx 180 ry 0 rz -180 deg; joints [1.651, 66.215, -28.516, 2.699, -37.73, -2.135]
  Call Extruder 0.01786
  MoveL (T19060) to (111.23, 120.16, 19.7) mm, rotated rx 180 ry 0 rz -180 deg; joints [1.875, 66.789, -29.593, 3.1, -37.236, -2.469]
  Call Extruder 0.04317
  MoveL (T19061) to (110.23, 121.16, 19.7) mm, rotated rx 180 ry 0 rz -180 deg; joints [1.875, 66.789, -29.593, 3.1, -37.236, -2.469]
  Call Extruder 0.01786
  MoveL (T19062) to (109.65, 121.16, 19.7) mm, rotated rx 180 ry 0 rz -180 deg; joints [1.875, 66.789, -29.593, 3.1, -37.236, -2.469]
  Call Extruder 0.04317
  MoveL (T19063) to (110.65, 120.16, 19.7) mm, rotated rx 180 ry 0 rz -180 deg; joints [1.875, 66.789, -29.593, 3.1, -37.236, -2.469]
  Call Extruder 0.01786
  MoveL (T19064) to (110.07, 120.16, 19.7) mm, rotated rx 180 ry 0 rz -180 deg; joints [1.875, 66.789, -29.593, 3.1, -37.236, -2.469]
  Call Extruder 0.04317
  MoveL (T19065) to (109.07, 121.16, 19.7) mm, rotated rx 180 ry 0 rz -180 deg; joints [1.875, 66.789, -29.593, 3.1, -37.236, -2.469]
  Call Extruder 0.01786
  MoveL (T19066) to (108.49, 121.16, 19.7) mm, rotated rx 180 ry 0 rz -180 deg; joints [1.875, 66.789, -29.593, 3.1, -37.236, -2.469]
  Call Extruder 0.04317
  MoveL (T19067) to (109.48, 120.16, 19.7) mm, rotated rx 180 ry 0 rz -180 deg; joints [1.875, 66.789, -29.593, 3.1, -37.236, -2.469]
  Call Extruder 0.01786
  MoveL (T19068) to (108.9, 120.16, 19.7) mm, rotated rx 180 ry 0 rz -180 deg; joints [1.875, 66.789, -29.593, 3.1, -37.236, -2.469]
  Call Extruder 0.04317
  MoveL (T19069) to (107.91, 121.16, 19.7) mm, rotated rx 180 ry 0 rz -180 deg; joints [1.796, 66.585, -29.21, 2.958, -37.412, -2.35]
  Call Extruder 0.01786
  MoveL (T19070) to (107.33, 121.16, 19.7) mm, rotated rx 180 ry 0 rz -180 deg; joints [1.796, 66.585, -29.21, 2.958, -37.412, -2.35]
  Call Extruder 0.04317
  MoveL (T19071) to (108.32, 120.16, 19.7) mm, rotated rx 180 ry 0 rz -180 deg; joints [1.796, 66.585, -29.21, 2.958, -37.412, -2.35]
  Call Extruder 0.01786
  MoveL (T19072) to (107.74, 120.16, 19.7) mm, rotated rx 180 ry 0 rz -180 deg; joints [1.796, 66.585, -29.21, 2.958, -37.412, -2.35]
  Call Extruder 0.04317
  MoveL (T19073) to (106.75, 121.16, 19.7) mm, rotated rx 180 ry 0 rz -180 deg; joints [1.796, 66.585, -29.21, 2.958, -37.412, -2.35]
  Call Extruder 0.01786
  MoveL (T19074) to (106.17, 121.16, 19.7) mm, rotated rx 180 ry 0 rz -180 deg; joints [1.796, 66.35, -29.174, 2.971, -37.213, -2.367]
  Call Extruder 0.06059
  MoveL (T19075) to (107.56, 119.76, 19.7) mm, rotated rx 180 ry 0 rz -180 deg; joints [3.301, 66.679, -29.792, 5.489, -37.014, -4.388]
  Call Extruder 0.01786
  MoveL (T19076) to (107.56, 119.18, 19.7) mm, rotated rx 180 ry 0 rz -180 deg; joints [3.301, 66.914, -29.828, 5.464, -37.212, -4.356]
  Call Extruder 0.08584
  MoveL (T19077) to (105.59, 121.16, 19.7) mm, rotated rx 180 ry 0 rz -180 deg; joints [3.301, 66.914, -29.828, 5.464, -37.212, -4.356]
  Call Extruder 0.01786
  MoveL (T19078) to (105.01, 121.16, 19.7) mm, rotated rx 180 ry 0 rz -180 deg; joints [3.301, 66.914, -29.828, 5.464, -37.212, -4.356]
  Call Extruder 0.1111
  MoveL (T19079) to (107.56, 118.6, 19.7) mm, rotated rx 180 ry 0 rz -180 deg; joints [3.301, 66.914, -29.828, 5.464, -37.212, -4.356]
  Call Extruder 0.01786
  MoveL (T19080) to (107.56, 118.02, 19.7) mm, rotated rx 180 ry 0 rz -180 deg; joints [3.301, 66.914, -29.828, 5.464, -37.212, -4.356]
  Call Extruder 0.13635
  MoveL (T19081) to (104.42, 121.16, 19.7) mm, rotated rx 180 ry 0 rz -180 deg; joints [3.301, 66.914, -29.828, 5.464, -37.212, -4.356]
  Call Extruder 0.01786
  MoveL (T19082) to (103.84, 121.16, 19.7) mm, rotated rx 180 ry 0 rz -180 deg; joints [3.301, 66.914, -29.828, 5.464, -37.212, -4.356]
  Call Extruder 0.1616
  MoveL (T19083) to (107.56, 117.44, 19.7) mm, rotated rx 180 ry 0 rz -180 deg; joints [3.301, 66.914, -29.828, 5.464, -37.212, -4.356]
  Call Extruder 0.01786
  MoveL (T19084) to (107.56, 116.86, 19.7) mm, rotated rx 180 ry 0 rz -180 deg; joints [3.301, 66.914, -29.828, 5.464, -37.212, -4.356]
  Call Extruder 0.1616
  MoveL (T19085) to (103.84, 120.58, 19.7) mm, rotated rx 180 ry 0 rz -180 deg; joints [3.301, 66.914, -29.828, 5.464, -37.212, -4.356]
  Call Extruder 0.01786
  MoveL (T19086) to (103.84, 119.99, 19.7) mm, rotated rx 180 ry 0 rz -180 deg; joints [3.316, 66.277, -28.632, 5.419, -37.769, -4.289]
  Call Extruder 0.29173
  MoveL (T19087) to (110.56, 113.28, 19.7) mm, rotated rx 180 ry 0 rz -180 deg; joints [3.316, 66.277, -28.632, 5.419, -37.769, -4.289]
  Call Extruder 0.01328
  MoveL (T19088) to (110.36, 112.9, 19.7) mm, rotated rx 180 ry 0 rz -180 deg; joints [3.316, 66.277, -28.632, 5.419, -37.769, -4.289]
  Call Extruder 0.2832
  MoveL (T19089) to (103.84, 119.41, 19.7) mm, rotated rx 180 ry 0 rz -180 deg; joints [1.863, 69.695, -35.051, 3.274, -34.688, -2.693]
  Call Extruder 0.01786
  MoveL (T19090) to (103.84, 118.83, 19.7) mm, rotated rx 180 ry 0 rz -180 deg; joints [1.863, 69.695, -35.051, 3.274, -34.688, -2.693]
  Call Extruder 0.27467
  MoveL (T19091) to (110.16, 112.51, 19.7) mm, rotated rx 180 ry 0 rz -180 deg; joints [1.863, 69.695, -35.051, 3.274, -34.688, -2.693]
  Call Extruder 0.01328
  MoveL (T19092) to (109.97, 112.13, 19.7) mm, rotated rx 180 ry 0 rz -180 deg; joints [1.861, 69.847, -35.336, 3.282, -34.555, -2.704]
  Call Extruder 0.26614
  MoveL (T19093) to (103.84, 118.25, 19.7) mm, rotated rx 180 ry 0 rz -180 deg; joints [1.861, 69.847, -35.336, 3.282, -34.555, -2.704]
  Call Extruder 0.01786
  MoveL (T19094) to (103.84, 117.67, 19.7) mm, rotated rx 180 ry 0 rz -180 deg; joints [1.861, 69.847, -35.336, 3.282, -34.555, -2.704]
  Call Extruder 0.25761
  MoveL (T19095) to (109.77, 111.74, 19.7) mm, rotated rx 180 ry 0 rz -180 deg; joints [1.915, 70.01, -35.641, 3.389, -34.415, -2.797]
  Call Extruder 0.01328
  MoveL (T19096) to (109.57, 111.36, 19.7) mm, rotated rx 180 ry 0 rz -180 deg; joints [1.915, 70.01, -35.641, 3.389, -34.415, -2.797]
  Call Extruder 0.24908
  MoveL (T19097) to (103.84, 117.09, 19.7) mm, rotated rx 180 ry 0 rz -180 deg; joints [1.915, 70.01, -35.641, 3.389, -34.415, -2.797]
  Call Extruder 0.01786
  MoveL (T19098) to (103.84, 116.51, 19.7) mm, rotated rx 180 ry 0 rz -180 deg; joints [1.803, 70.309, -36.204, 3.213, -34.147, -2.66]
  Call Extruder 0.24055
  MoveL (T19099) to (109.38, 110.97, 19.7) mm, rotated rx 180 ry 0 rz -180 deg; joints [1.803, 70.309, -36.204, 3.213, -34.147, -2.66]
  Call Extruder 0.01328
  MoveL (T19100) to (109.18, 110.59, 19.7) mm, rotated rx 180 ry 0 rz -180 deg; joints [1.794, 70.369, -36.317, 3.201, -34.094, -2.651]
  Call Extruder 0.23202
  MoveL (T19101) to (103.84, 115.93, 19.7) mm, rotated rx 180 ry 0 rz -180 deg; joints [1.794, 70.369, -36.317, 3.201, -34.094, -2.651]
  Call Extruder 0.01786
  MoveL (T19102) to (103.84, 115.35, 19.7) mm, rotated rx 180 ry 0 rz -180 deg; joints [1.794, 70.369, -36.317, 3.201, -34.094, -2.651]
  Call Extruder 0.22349
  MoveL (T19103) to (108.98, 110.21, 19.7) mm, rotated rx 180 ry 0 rz -180 deg; joints [1.787, 70.998, -37.498, 3.235, -33.542, -2.697]
  Call Extruder 0.01328
  MoveL (T19104) to (108.79, 109.82, 19.7) mm, rotated rx 180 ry 0 rz -180 deg; joints [1.787, 70.998, -37.498, 3.235, -33.542, -2.697]
  Call Extruder 0.21496
  MoveL (T19105) to (103.84, 114.77, 19.7) mm, rotated rx 180 ry 0 rz -180 deg; joints [1.787, 70.998, -37.498, 3.235, -33.542, -2.697]
  Call Extruder 0.01786
  MoveL (T19106) to (103.84, 114.18, 19.7) mm, rotated rx 180 ry 0 rz -180 deg; joints [1.763, 70.996, -37.494, 3.191, -33.543, -2.661]
  Call Extruder 0.20642
  MoveL (T19107) to (108.59, 109.44, 19.7) mm, rotated rx 180 ry 0 rz -180 deg; joints [1.763, 70.996, -37.494, 3.191, -33.543, -2.661]
  Call Extruder 0.01328
  MoveL (T19108) to (108.4, 109.05, 19.7) mm, rotated rx 180 ry 0 rz -180 deg; joints [1.763, 70.996, -37.494, 3.191, -33.543, -2.661]
  Call Extruder 0.19789
  MoveL (T19109) to (103.84, 113.6, 19.7) mm, rotated rx 180 ry 0 rz -180 deg; joints [1.659, 70.669, -36.88, 2.98, -33.825, -2.477]
  Call Extruder 0.01786
  MoveL (T19110) to (103.84, 113.02, 19.7) mm, rotated rx 180 ry 0 rz -180 deg; joints [1.659, 70.669, -36.88, 2.98, -33.825, -2.477]
  Call Extruder 0.18936
  MoveL (T19111) to (108.2, 108.67, 19.7) mm, rotated rx 180 ry 0 rz -180 deg; joints [1.659, 70.669, -36.88, 2.98, -33.825, -2.477]
  Call Extruder 0.01328
  MoveL (T19112) to (108, 108.28, 19.7) mm, rotated rx 180 ry 0 rz -180 deg; joints [1.628, 70.754, -37.039, 2.931, -33.749, -2.438]
  Call Extruder 0.18083
  MoveL (T19113) to (103.84, 112.44, 19.7) mm, rotated rx 180 ry 0 rz -180 deg; joints [1.628, 70.754, -37.039, 2.931, -33.749, -2.438]
  Call Extruder 0.01786
  MoveL (T19114) to (103.84, 111.86, 19.7) mm, rotated rx 180 ry 0 rz -180 deg; joints [1.628, 70.754, -37.039, 2.931, -33.749, -2.438]
  Call Extruder 0.1723
  MoveL (T19115) to (107.81, 107.9, 19.7) mm, rotated rx 180 ry 0 rz -180 deg; joints [1.607, 70.778, -37.084, 2.894, -33.727, -2.408]
  Call Extruder 0.01328
  MoveL (T19116) to (107.61, 107.51, 19.7) mm, rotated rx 180 ry 0 rz -180 deg; joints [1.607, 70.778, -37.084, 2.894, -33.727, -2.408]
  Call Extruder 0.16377
  MoveL (T19117) to (103.84, 111.28, 19.7) mm, rotated rx 180 ry 0 rz -180 deg; joints [1.607, 70.778, -37.084, 2.894, -33.727, -2.408]
  Call Extruder 0.01786
  MoveL (T19118) to (103.84, 110.7, 19.7) mm, rotated rx 180 ry 0 rz -180 deg; joints [1.467, 70.767, -37.064, 2.642, -33.731, -2.197]
  Call Extruder 0.15795
  MoveL (T19119) to (107.48, 107.07, 19.7) mm, rotated rx 180 ry 0 rz -180 deg; joints [1.467, 70.767, -37.064, 2.642, -33.731, -2.197]
  Call Extruder 0.01786
  MoveL (T19120) to (107.48, 106.48, 19.7) mm, rotated rx 180 ry 0 rz -180 deg; joints [1.467, 70.767, -37.064, 2.642, -33.731, -2.197]
  Call Extruder 0.15795
  MoveL (T19121) to (103.84, 110.12, 19.7) mm, rotated rx 180 ry 0 rz -180 deg; joints [1.396, 70.966, -37.437, 2.526, -33.554, -2.106]
  Call Extruder 0.01786
  MoveL (T19122) to (103.84, 109.54, 19.7) mm, rotated rx 180 ry 0 rz -180 deg; joints [1.396, 70.966, -37.437, 2.526, -33.554, -2.106]
  Call Extruder 0.16591
  MoveL (T19123) to (107.66, 105.72, 19.7) mm, rotated rx 180 ry 0 rz -180 deg; joints [1.652, 70.986, -37.476, 2.991, -33.546, -2.494]
  Set speed (45.0 mm/s)
  Call Extruder -1.6
  MoveL (T19124) to (107.66, 105.72, 19.7) mm, rotated rx 180 ry 0 rz -180 deg; joints [1.652, 70.986, -37.476, 2.991, -33.546, -2.494]
  Set speed (120.0 mm/s)
  MoveL (T19125) to (107.66, 105.72, 19.7) mm, rotated rx 180 ry 0 rz -180 deg; joints [1.652, 70.986, -37.476, 2.991, -33.546, -2.494]
  Call Extruder -0.38
  MoveL (T19126) to (106.91, 106.47, 19.7) mm, rotated rx 180 ry 0 rz -180 deg; joints [1.652, 70.986, -37.476, 2.991, -33.546, -2.494]
  Set speed (45.0 mm/s)
  Call Extruder -0.02
  MoveL (T19127) to (106.91, 106.47, 19.7) mm, rotated rx 180 ry 0 rz -180 deg; joints [1.652, 70.986, -37.476, 2.991, -33.546, -2.494]
  Set speed (150.0 mm/s)
  MoveL (T19128) to (106.91, 106.47, 21.7) mm, rotated rx 180 ry 0 rz -180 deg; joints [1.652, 70.986, -37.476, 2.991, -33.546, -2.494]
  MoveL (T19129) to (109.14, 103.66, 21.7) mm, rotated rx 180 ry 0 rz -180 deg; joints [1.652, 70.986, -37.476, 2.991, -33.546, -2.494]
  MoveL (T19130) to (109.14, 103.66, 19.7) mm, rotated rx 180 ry 0 rz -180 deg; joints [1.54, 70.977, -37.458, 2.788, -33.55, -2.324]
  Set speed (40.0 mm/s)
  Call Extruder 2.0
  MoveL (T19131) to (109.14, 103.66, 19.7) mm, rotated rx 180 ry 0 rz -180 deg; joints [1.54, 70.977, -37.458, 2.788, -33.55, -2.324]
  Call Extruder 0.23019
  MoveL (T19132) to (103.84, 108.96, 19.7) mm, rotated rx 180 ry 0 rz -180 deg; joints [1.54, 70.977, -37.458, 2.788, -33.55, -2.324]
  Call Extruder 0.01786
  MoveL (T19133) to (103.84, 108.38, 19.7) mm, rotated rx 180 ry 0 rz -180 deg; joints [1.54, 70.977, -37.458, 2.788, -33.55, -2.324]
  Call Extruder 0.19697
  MoveL (T19134) to (108.38, 103.84, 19.7) mm, rotated rx 180 ry 0 rz -180 deg; joints [1.54, 70.977, -37.458, 2.788, -33.55, -2.324]
  Call Extruder 0.01786
  MoveL (T19135) to (107.79, 103.84, 19.7) mm, rotated rx 180 ry 0 rz -180 deg; joints [1.54, 70.977, -37.458, 2.788, -33.55, -2.324]
  Call Extruder 0.17171
  MoveL (T19136) to (103.84, 107.79, 19.7) mm, rotated rx 180 ry 0 rz -180 deg; joints [1.54, 70.977, -37.458, 2.788, -33.55, -2.324]
  Call Extruder 0.01786
  MoveL (T19137) to (103.84, 107.21, 19.7) mm, rotated rx 180 ry 0 rz -180 deg; joints [1.54, 70.744, -37.416, 2.802, -33.36, -2.341]
  Call Extruder 0.14646
  MoveL (T19138) to (107.21, 103.84, 19.7) mm, rotated rx 180 ry 0 rz -180 deg; joints [1.407, 65.981, -28.484, 2.311, -37.52, -1.833]
  Call Extruder 0.01786
  MoveL (T19139) to (106.63, 103.84, 19.7) mm, rotated rx 180 ry 0 rz -180 deg; joints [1.407, 66.193, -28.516, 2.302, -37.7, -1.822]
  Call Extruder 0.1212
  MoveL (T19140) to (103.84, 106.63, 19.7) mm, rotated rx 180 ry 0 rz -180 deg; joints [1.407, 66.193, -28.516, 2.302, -37.7, -1.822]
  Call Extruder 0.01786
  MoveL (T19141) to (103.84, 106.05, 19.7) mm, rotated rx 180 ry 0 rz -180 deg; joints [1.407, 66.193, -28.516, 2.302, -37.7, -1.822]
  Call Extruder 0.09595
  MoveL (T19142) to (106.05, 103.84, 19.7) mm, rotated rx 180 ry 0 rz -180 deg; joints [1.407, 66.193, -28.516, 2.302, -37.7, -1.822]
  Call Extruder 0.01786
  MoveL (T19143) to (105.47, 103.84, 19.7) mm, rotated rx 180 ry 0 rz -180 deg; joints [1.407, 66.193, -28.516, 2.302, -37.7, -1.822]
  Call Extruder 0.07069
  MoveL (T19144) to (103.84, 105.47, 19.7) mm, rotated rx 180 ry 0 rz -180 deg; joints [1.407, 66.193, -28.516, 2.302, -37.7, -1.822]
  Call Extruder 0.01786
  MoveL (T19145) to (103.84, 104.89, 19.7) mm, rotated rx 180 ry 0 rz -180 deg; joints [1.407, 66.193, -28.516, 2.302, -37.7, -1.822]
  Call Extruder 0.04544
  MoveL (T19146) to (104.89, 103.84, 19.7) mm, rotated rx 180 ry 0 rz -180 deg; joints [1.407, 66.193, -28.516, 2.302, -37.7, -1.822]
  Call Extruder 0.01786
  MoveL (T19147) to (104.31, 103.84, 19.7) mm, rotated rx 180 ry 0 rz -180 deg; joints [1.407, 66.193, -28.516, 2.302, -37.7, -1.822]
  Call Extruder 0.02815
  MoveL (T19148) to (103.66, 104.49, 19.7) mm, rotated rx 180 ry 0 rz -180 deg; joints [1.407, 66.193, -28.516, 2.302, -37.7, -1.822]
  Set speed (45.0 mm/s)
  Call Extruder -1.6
  MoveL (T19149) to (103.66, 104.49, 19.7) mm, rotated rx 180 ry 0 rz -180 deg; joints [1.407, 66.193, -28.516, 2.302, -37.7, -1.822]
  Set speed (120.0 mm/s)
  MoveL (T19150) to (103.66, 104.49, 19.7) mm, rotated rx 180 ry 0 rz -180 deg; joints [1.363, 71.036, -37.608, 2.473, -33.452, -2.064]
  Call Extruder -0.3262
  MoveL (T19151) to (104.31, 103.84, 19.7) mm, rotated rx 180 ry 0 rz -180 deg; joints [1.363, 71.036, -37.608, 2.473, -33.452, -2.064]
  Call Extruder -0.0538
  MoveL (T19152) to (104.46, 103.84, 19.7) mm, rotated rx 180 ry 0 rz -180 deg; joints [1.363, 71.036, -37.608, 2.473, -33.452, -2.064]
  Set speed (45.0 mm/s)
  Call Extruder -0.02
  MoveL (T19153) to (104.46, 103.84, 19.7) mm, rotated rx 180 ry 0 rz -180 deg; joints [3.241, 71.263, -38.035, 5.901, -33.368, -4.933]
  Set speed (150.0 mm/s)
  MoveL (T19154) to (104.46, 103.84, 21.7) mm, rotated rx 180 ry 0 rz -180 deg; joints [3.241, 71.263, -38.035, 5.901, -33.368, -4.933]
  MoveL (T19155) to (109.4, 105.47, 21.7) mm, rotated rx 180 ry 0 rz -180 deg; joints [3.351, 66.179, -28.489, 5.471, -37.817, -4.327]
  MoveL (T19156) to (109.4, 105.47, 19.9) mm, rotated rx 180 ry 0 rz -180 deg; joints [3.351, 66.179, -28.489, 5.471, -37.817, -4.327]
  Set speed (40.0 mm/s)
  Call Extruder 2.0
  MoveL (T19157) to (109.4, 105.47, 19.9) mm, rotated rx 180 ry 0 rz -180 deg; joints [3.351, 66.179, -28.489, 5.471, -37.817, -4.327]
  Call Extruder 0.25145
  MoveL (T19158) to (117.65, 105.47, 19.9) mm, rotated rx 180 ry 0 rz -180 deg; joints [3.351, 66.179, -28.489, 5.471, -37.817, -4.327]
  Call Extruder 0.10939
  MoveL (T19159) to (117.65, 109.06, 19.9) mm, rotated rx 180 ry 0 rz -180 deg; joints [1.409, 65.988, -28.13, 2.296, -37.88, -1.812]
  Call Extruder 0.14732
  MoveL (T19160) to (112.81, 109.06, 19.9) mm, rotated rx 180 ry 0 rz -180 deg; joints [1.409, 65.988, -28.13, 2.296, -37.88, -1.812]
  Call Extruder 0.31102
  MoveL (T19161) to (117.47, 118.15, 19.9) mm, rotated rx 180 ry 0 rz -180 deg; joints [1.409, 65.988, -28.13, 2.296, -37.88, -1.812]
  Call Extruder 0.05209
  MoveL (T19162) to (117.47, 119.86, 19.9) mm, rotated rx 180 ry 0 rz -180 deg; joints [1.409, 65.988, -28.13, 2.296, -37.88, -1.812]
  Call Extruder 0.29244
  MoveL (T19163) to (107.87, 119.86, 19.9) mm, rotated rx 180 ry 0 rz -180 deg; joints [1.407, 66.178, -28.487, 2.301, -37.714, -1.821]
  Call Extruder 0.10939
  MoveL (T19164) to (107.87, 116.27, 19.9) mm, rotated rx 180 ry 0 rz -180 deg; joints [1.407, 66.178, -28.487, 2.301, -37.714, -1.821]
  Call Extruder 0.13869
  MoveL (T19165) to (112.42, 116.27, 19.9) mm, rotated rx 180 ry 0 rz -180 deg; joints [1.407, 66.178, -28.487, 2.301, -37.714, -1.821]
  Call Extruder 0.31084
  MoveL (T19166) to (107.78, 107.18, 19.9) mm, rotated rx 180 ry 0 rz -180 deg; joints [1.365, 65.984, -28.122, 2.224, -37.882, -1.756]
  Call Extruder 0.05206
  MoveL (T19167) to (107.78, 105.47, 19.9) mm, rotated rx 180 ry 0 rz -180 deg; joints [1.365, 65.984, -28.122, 2.224, -37.882, -1.756]
  Call Extruder 0.04735
  MoveL (T19168) to (109.34, 105.47, 19.9) mm, rotated rx 180 ry 0 rz -180 deg; joints [1.365, 65.984, -28.122, 2.224, -37.882, -1.756]
  Set speed (150.0 mm/s)
  MoveL (T19169) to (109, 105.88, 19.9) mm, rotated rx 180 ry 0 rz -180 deg; joints [1.365, 65.984, -28.122, 2.224, -37.882, -1.756]
  Set speed (40.0 mm/s)
  MoveL (T19170) to (109, 105.88, 19.9) mm, rotated rx 180 ry 0 rz -180 deg; joints [1.365, 65.984, -28.122, 2.224, -37.882, -1.756]
  Call Extruder 0.25124
  MoveL (T19171) to (117.24, 105.88, 19.9) mm, rotated rx 180 ry 0 rz -180 deg; joints [1.319, 71.161, -37.843, 2.401, -33.341, -2.006]
  Call Extruder 0.08459
  MoveL (T19172) to (117.24, 108.65, 19.9) mm, rotated rx 180 ry 0 rz -180 deg; joints [1.319, 71.161, -37.843, 2.401, -33.341, -2.006]
  Call Extruder 0.1552
  MoveL (T19173) to (112.15, 108.65, 19.9) mm, rotated rx 180 ry 0 rz -180 deg; joints [1.319, 71.161, -37.843, 2.401, -33.341, -2.006]
  Call Extruder 0.32831
  MoveL (T19174) to (117.06, 118.25, 19.9) mm, rotated rx 180 ry 0 rz -180 deg; joints [3.282, 71.399, -38.291, 5.992, -33.252, -5.017]
  Call Extruder 0.0367
  MoveL (T19175) to (117.06, 119.45, 19.9) mm, rotated rx 180 ry 0 rz -180 deg; joints [3.398, 66.081, -28.305, 5.536, -37.906, -4.373]
  Call Extruder 0.26763
  MoveL (T19176) to (108.27, 119.45, 19.9) mm, rotated rx 180 ry 0 rz -180 deg; joints [3.398, 66.081, -28.305, 5.536, -37.906, -4.373]
  Call Extruder 0.08459
  MoveL (T19177) to (108.27, 116.67, 19.9) mm, rotated rx 180 ry 0 rz -180 deg; joints [3.398, 66.081, -28.305, 5.536, -37.906, -4.373]
  Call Extruder 0.14654
  MoveL (T19178) to (113.08, 116.67, 19.9) mm, rotated rx 180 ry 0 rz -180 deg; joints [3.398, 66.081, -28.305, 5.536, -37.906, -4.373]
  Call Extruder 0.32811
  MoveL (T19179) to (108.19, 107.08, 19.9) mm, rotated rx 180 ry 0 rz -180 deg; joints [1.366, 65.882, -27.931, 2.221, -37.972, -1.751]
  Call Extruder 0.03668
  MoveL (T19180) to (108.19, 105.88, 19.9) mm, rotated rx 180 ry 0 rz -180 deg; joints [1.366, 65.882, -27.931, 2.221, -37.972, -1.751]
  Call Extruder 0.02276
  MoveL (T19181) to (108.94, 105.88, 19.9) mm, rotated rx 180 ry 0 rz -180 deg; joints [1.366, 65.882, -27.931, 2.221, -37.972, -1.751]
  Set speed (150.0 mm/s)
  MoveL (T19182) to (108.6, 106.28, 19.9) mm, rotated rx 180 ry 0 rz -180 deg; joints [1.366, 65.882, -27.931, 2.221, -37.972, -1.751]
  Set speed (25.0 mm/s)
  MoveL (T19183) to (108.6, 106.28, 19.9) mm, rotated rx 180 ry 0 rz -180 deg; joints [1.365, 65.968, -28.093, 2.223, -37.896, -1.755]
  Call Extruder 0.25102
  MoveL (T19184) to (116.84, 106.28, 19.9) mm, rotated rx 180 ry 0 rz -180 deg; joints [1.365, 65.968, -28.093, 2.223, -37.896, -1.755]
  Call Extruder 0.05979
  MoveL (T19185) to (116.84, 108.25, 19.9) mm, rotated rx 180 ry 0 rz -180 deg; joints [1.332, 65.776, -27.733, 2.161, -38.063, -1.702]
  Call Extruder 0.16307
  MoveL (T19186) to (111.48, 108.25, 19.9) mm, rotated rx 180 ry 0 rz -180 deg; joints [1.332, 65.776, -27.733, 2.161, -38.063, -1.702]
  Call Extruder 0.3456
  MoveL (T19187) to (116.65, 118.34, 19.9) mm, rotated rx 180 ry 0 rz -180 deg; joints [1.332, 65.776, -27.733, 2.161, -38.063, -1.702]
  Call Extruder 0.02131
  MoveL (T19188) to (116.65, 119.04, 19.9) mm, rotated rx 180 ry 0 rz -180 deg; joints [1.332, 65.776, -27.733, 2.161, -38.063, -1.702]
  Call Extruder 0.24283
  MoveL (T19189) to (108.68, 119.04, 19.9) mm, rotated rx 180 ry 0 rz -180 deg; joints [1.332, 65.776, -27.733, 2.161, -38.063, -1.702]
  Call Extruder 0.05979
  MoveL (T19190) to (108.68, 117.08, 19.9) mm, rotated rx 180 ry 0 rz -180 deg; joints [1.332, 65.776, -27.733, 2.161, -38.063, -1.702]
  Call Extruder 0.15438
  MoveL (T19191) to (113.75, 117.08, 19.9) mm, rotated rx 180 ry 0 rz -180 deg; joints [1.323, 65.776, -27.732, 2.146, -38.063, -1.69]
  Call Extruder 0.34538
  MoveL (T19192) to (108.6, 106.98, 19.9) mm, rotated rx 180 ry 0 rz -180 deg; joints [1.276, 71.286, -38.079, 2.329, -33.229, -1.948]
  Call Extruder 0.01947
  MoveL (T19193) to (108.6, 106.34, 19.9) mm, rotated rx 180 ry 0 rz -180 deg; joints [1.276, 71.286, -38.079, 2.329, -33.229, -1.948]
  Set speed (150.0 mm/s)
  MoveL (T19194) to (108.54, 105.89, 19.9) mm, rotated rx 180 ry 0 rz -180 deg; joints [1.276, 71.286, -38.079, 2.329, -33.229, -1.948]
  Set speed (45.0 mm/s)
  Call Extruder -1.6
  MoveL (T19195) to (108.54, 105.89, 19.9) mm, rotated rx 180 ry 0 rz -180 deg; joints [3.322, 71.537, -38.55, 6.085, -33.135, -5.101]
  Set speed (120.0 mm/s)
  MoveL (T19196) to (108.54, 105.89, 19.9) mm, rotated rx 180 ry 0 rz -180 deg; joints [3.322, 71.537, -38.55, 6.085, -33.135, -5.101]
  Call Extruder -0.38
  MoveL (T19197) to (109.66, 106.33, 19.9) mm, rotated rx 180 ry 0 rz -180 deg; joints [3.322, 71.537, -38.55, 6.085, -33.135, -5.101]
  Set speed (45.0 mm/s)
  Call Extruder -0.02
  MoveL (T19198) to (109.66, 106.33, 19.9) mm, rotated rx 180 ry 0 rz -180 deg; joints [3.445, 65.983, -28.121, 5.601, -37.995, -4.419]
  Set speed (150.0 mm/s)
  MoveL (T19199) to (109.66, 106.33, 21.9) mm, rotated rx 180 ry 0 rz -180 deg; joints [3.445, 65.983, -28.121, 5.601, -37.995, -4.419]
  MoveL (T19200) to (104.34, 103.54, 21.9) mm, rotated rx 180 ry 0 rz -180 deg; joints [3.445, 65.983, -28.121, 5.601, -37.995, -4.419]
  MoveL (T19201) to (104.34, 103.54, 19.9) mm, rotated rx 180 ry 0 rz -180 deg; joints [1.339, 65.776, -27.733, 2.172, -38.063, -1.71]
  Set speed (40.0 mm/s)
  Call Extruder 2.0
  MoveL (T19202) to (104.34, 103.54, 19.9) mm, rotated rx 180 ry 0 rz -180 deg; joints [1.339, 65.776, -27.733, 2.172, -38.063, -1.71]
  Call Extruder 0.52159
  MoveL (T19203) to (121.46, 103.54, 19.9) mm, rotated rx 180 ry 0 rz -180 deg; joints [1.339, 65.776, -27.733, 2.172, -38.063, -1.71]
  Call Extruder 0.54596
  MoveL (T19204) to (121.46, 121.46, 19.9) mm, rotated rx 180 ry 0 rz -180 deg; joints [1.326, 65.791, -27.761, 2.151, -38.05, -1.694]
  Call Extruder 0.54596
  MoveL (T19205) to (103.54, 121.46, 19.9) mm, rotated rx 180 ry 0 rz -180 deg; joints [1.326, 65.791, -27.761, 2.151, -38.05, -1.694]
  Call Extruder 0.54596
  MoveL (T19206) to (103.54, 103.54, 19.9) mm, rotated rx 180 ry 0 rz -180 deg; joints [1.326, 65.791, -27.761, 2.151, -38.05, -1.694]
  Call Extruder 0.02254
  MoveL (T19207) to (104.28, 103.54, 19.9) mm, rotated rx 180 ry 0 rz -180 deg; joints [1.326, 65.791, -27.761, 2.151, -38.05, -1.694]
  Set speed (150.0 mm/s)
  MoveL (T19208) to (103.53, 103.13, 19.9) mm, rotated rx 180 ry 0 rz -180 deg; joints [1.326, 65.791, -27.761, 2.151, -38.05, -1.694]
  Set speed (40.0 mm/s)
  MoveL (T19209) to (103.53, 103.13, 19.9) mm, rotated rx 180 ry 0 rz -180 deg; joints [1.326, 65.791, -27.761, 2.151, -38.05, -1.694]
  Call Extruder 0.55858
  MoveL (T19210) to (121.87, 103.13, 19.9) mm, rotated rx 180 ry 0 rz -180 deg; joints [1.326, 65.791, -27.761, 2.151, -38.05, -1.694]
  Call Extruder 0.57077
  MoveL (T19211) to (121.87, 121.87, 19.9) mm, rotated rx 180 ry 0 rz -180 deg; joints [1.326, 65.791, -27.761, 2.151, -38.05, -1.694]
  Call Extruder 0.57077
  MoveL (T19212) to (103.13, 121.87, 19.9) mm, rotated rx 180 ry 0 rz -180 deg; joints [1.326, 65.791, -27.761, 2.151, -38.05, -1.694]
  Call Extruder 0.57077
  MoveL (T19213) to (103.13, 103.13, 19.9) mm, rotated rx 180 ry 0 rz -180 deg; joints [1.326, 65.791, -27.761, 2.151, -38.05, -1.694]
  Call Extruder 0.01036
  MoveL (T19214) to (103.47, 103.13, 19.9) mm, rotated rx 180 ry 0 rz -180 deg; joints [1.323, 65.776, -27.732, 2.146, -38.063, -1.69]
  Set speed (150.0 mm/s)
  MoveL (T19215) to (102.72, 102.81, 19.9) mm, rotated rx 180 ry 0 rz -180 deg; joints [1.323, 65.776, -27.732, 2.146, -38.063, -1.69]
  Set speed (25.0 mm/s)
  MoveL (T19216) to (102.72, 102.81, 19.9) mm, rotated rx 180 ry 0 rz -180 deg; joints [1.323, 65.776, -27.732, 2.146, -38.063, -1.69]
  Call Extruder 0.00259
  MoveL (T19217) to (102.72, 102.72, 19.9) mm, rotated rx 180 ry 0 rz -180 deg; joints [1.323, 65.776, -27.732, 2.146, -38.063, -1.69]
  Call Extruder 0.59557
  MoveL (T19218) to (122.28, 102.72, 19.9) mm, rotated rx 180 ry 0 rz -180 deg; joints [1.321, 66.011, -28.173, 2.153, -37.857, -1.7]
  Call Extruder 0.59557
  MoveL (T19219) to (122.28, 122.28, 19.9) mm, rotated rx 180 ry 0 rz -180 deg; joints [1.321, 66.011, -28.173, 2.153, -37.857, -1.7]
  Call Extruder 0.59557
  MoveL (T19220) to (102.72, 122.28, 19.9) mm, rotated rx 180 ry 0 rz -180 deg; joints [1.321, 66.011, -28.173, 2.153, -37.857, -1.7]
  Call Extruder 0.59115
  MoveL (T19221) to (102.72, 102.87, 19.9) mm, rotated rx 180 ry 0 rz -180 deg; joints [1.321, 66.011, -28.173, 2.153, -37.857, -1.7]
  Set speed (150.0 mm/s)
  MoveL (T19222) to (102.78, 102.75, 19.9) mm, rotated rx 180 ry 0 rz -180 deg; joints [1.321, 66.011, -28.173, 2.153, -37.857, -1.7]
  Set speed (45.0 mm/s)
  Call Extruder -1.6
  MoveL (T19223) to (102.78, 102.75, 19.9) mm, rotated rx 180 ry 0 rz -180 deg; joints [1.707, 66.085, -28.313, 2.785, -37.805, -2.201]
  Set speed (120.0 mm/s)
  MoveL (T19224) to (102.78, 102.75, 19.9) mm, rotated rx 180 ry 0 rz -180 deg; joints [1.707, 66.085, -28.313, 2.785, -37.805, -2.201]
  Call Extruder -0.05166
  MoveL (T19225) to (102.72, 102.72, 19.9) mm, rotated rx 180 ry 0 rz -180 deg; joints [1.707, 66.085, -28.313, 2.785, -37.805, -2.201]
  Call Extruder -0.32834
  MoveL (T19226) to (103.65, 102.72, 19.9) mm, rotated rx 180 ry 0 rz -180 deg; joints [1.707, 66.085, -28.313, 2.785, -37.805, -2.201]
  Set speed (45.0 mm/s)
  Call Extruder -0.02
  MoveL (T19227) to (103.65, 102.72, 19.9) mm, rotated rx 180 ry 0 rz -180 deg; joints [1.707, 66.085, -28.313, 2.785, -37.805, -2.201]
  Set speed (150.0 mm/s)
  MoveL (T19228) to (103.65, 102.72, 21.9) mm, rotated rx 180 ry 0 rz -180 deg; joints [1.707, 66.085, -28.313, 2.785, -37.805, -2.201]
  MoveL (T19229) to (120.51, 103.66, 21.9) mm, rotated rx 180 ry 0 rz -180 deg; joints [1.707, 66.085, -28.313, 2.785, -37.805, -2.201]
  MoveL (T19230) to (120.51, 103.66, 19.9) mm, rotated rx 180 ry 0 rz -180 deg; joints [1.442, 66.068, -28.281, 2.352, -37.811, -1.859]
  Set speed (40.0 mm/s)
  Call Extruder 2.0
  MoveL (T19231) to (120.51, 103.66, 19.9) mm, rotated rx 180 ry 0 rz -180 deg; joints [1.442, 66.068, -28.281, 2.352, -37.811, -1.859]
  Call Extruder 0.02815
  MoveL (T19232) to (121.16, 104.31, 19.9) mm, rotated rx 180 ry 0 rz -180 deg; joints [1.657, 66.083, -28.309, 2.704, -37.805, -2.137]
  Call Extruder 0.01786
  MoveL (T19233) to (121.16, 104.89, 19.9) mm, rotated rx 180 ry 0 rz -180 deg; joints [1.657, 66.083, -28.309, 2.704, -37.805, -2.137]
  Call Extruder 0.04544
  MoveL (T19234) to (120.11, 103.84, 19.9) mm, rotated rx 180 ry 0 rz -180 deg; joints [1.679, 66.106, -28.352, 2.74, -37.786, -2.166]
  Call Extruder 0.01786
  MoveL (T19235) to (119.53, 103.84, 19.9) mm, rotated rx 180 ry 0 rz -180 deg; joints [1.679, 66.106, -28.352, 2.74, -37.786, -2.166]
  Call Extruder 0.0707
  MoveL (T19236) to (121.16, 105.47, 19.9) mm, rotated rx 180 ry 0 rz -180 deg; joints [1.679, 66.106, -28.352, 2.74, -37.786, -2.166]
  Call Extruder 0.01786
  MoveL (T19237) to (121.16, 106.05, 19.9) mm, rotated rx 180 ry 0 rz -180 deg; joints [1.743, 66.268, -28.655, 2.854, -37.647, -2.26]
  Call Extruder 0.09595
  MoveL (T19238) to (118.95, 103.84, 19.9) mm, rotated rx 180 ry 0 rz -180 deg; joints [1.743, 66.268, -28.655, 2.854, -37.647, -2.26]
  Call Extruder 0.01786
  MoveL (T19239) to (118.37, 103.84, 19.9) mm, rotated rx 180 ry 0 rz -180 deg; joints [1.743, 66.268, -28.655, 2.854, -37.647, -2.26]
  Call Extruder 0.12121
  MoveL (T19240) to (121.16, 106.63, 19.9) mm, rotated rx 180 ry 0 rz -180 deg; joints [1.821, 66.094, -28.329, 2.971, -37.802, -2.348]
  Call Extruder 0.01786
  MoveL (T19241) to (121.16, 107.21, 19.9) mm, rotated rx 180 ry 0 rz -180 deg; joints [1.821, 66.094, -28.329, 2.971, -37.802, -2.348]
  Call Extruder 0.14646
  MoveL (T19242) to (117.79, 103.84, 19.9) mm, rotated rx 180 ry 0 rz -180 deg; joints [1.941, 66.103, -28.346, 3.168, -37.799, -2.504]
  Call Extruder 0.01786
  MoveL (T19243) to (117.21, 103.84, 19.9) mm, rotated rx 180 ry 0 rz -180 deg; joints [1.941, 66.103, -28.346, 3.168, -37.799, -2.504]
  Call Extruder 0.17172
  MoveL (T19244) to (121.16, 107.79, 19.9) mm, rotated rx 180 ry 0 rz -180 deg; joints [1.941, 66.103, -28.346, 3.168, -37.799, -2.504]
  Call Extruder 0.01786
  MoveL (T19245) to (121.16, 108.38, 19.9) mm, rotated rx 180 ry 0 rz -180 deg; joints [3.239, 69.755, -35.202, 5.697, -34.685, -4.69]
  Call Extruder 0.19697
  MoveL (T19246) to (116.62, 103.84, 19.9) mm, rotated rx 180 ry 0 rz -180 deg; joints [3.239, 69.755, -35.202, 5.697, -34.685, -4.69]
  Call Extruder 0.01786
  MoveL (T19247) to (116.04, 103.84, 19.9) mm, rotated rx 180 ry 0 rz -180 deg; joints [3.239, 69.755, -35.202, 5.697, -34.685, -4.69]
  Call Extruder 0.0573
  MoveL (T19248) to (117.36, 105.16, 19.9) mm, rotated rx 180 ry 0 rz -180 deg; joints [3.232, 70.086, -35.825, 5.728, -34.395, -4.731]
  Call Extruder 0.01786
  MoveL (T19249) to (116.78, 105.16, 19.9) mm, rotated rx 180 ry 0 rz -180 deg; joints [3.232, 70.086, -35.825, 5.728, -34.395, -4.731]
  Call Extruder 0.0573
  MoveL (T19250) to (115.46, 103.84, 19.9) mm, rotated rx 180 ry 0 rz -180 deg; joints [2.845, 71.103, -37.734, 5.163, -33.476, -4.31]
  Call Extruder 0.01786
  MoveL (T19251) to (114.88, 103.84, 19.9) mm, rotated rx 180 ry 0 rz -180 deg; joints [2.845, 71.103, -37.734, 5.163, -33.476, -4.31]
  Call Extruder 0.0573
  MoveL (T19252) to (116.2, 105.16, 19.9) mm, rotated rx 180 ry 0 rz -180 deg; joints [2.845, 71.103, -37.734, 5.163, -33.476, -4.31]
  Call Extruder 0.01786
  MoveL (T19253) to (115.62, 105.16, 19.9) mm, rotated rx 180 ry 0 rz -180 deg; joints [3.211, 71.161, -37.844, 5.832, -33.454, -4.871]
  Call Extruder 0.0573
  MoveL (T19254) to (114.3, 103.84, 19.9) mm, rotated rx 180 ry 0 rz -180 deg; joints [3.211, 71.161, -37.844, 5.832, -33.454, -4.871]
  Call Extruder 0.01786
  MoveL (T19255) to (113.72, 103.84, 19.9) mm, rotated rx 180 ry 0 rz -180 deg; joints [3.211, 71.161, -37.844, 5.832, -33.454, -4.871]
  Call Extruder 0.0573
  MoveL (T19256) to (115.04, 105.16, 19.9) mm, rotated rx 180 ry 0 rz -180 deg; joints [3.211, 71.161, -37.844, 5.832, -33.454, -4.871]
  Call Extruder 0.01786
  MoveL (T19257) to (114.46, 105.16, 19.9) mm, rotated rx 180 ry 0 rz -180 deg; joints [1.893, 67.23, -30.46, 3.16, -36.811, -2.531]
  Call Extruder 0.0573
  MoveL (T19258) to (113.14, 103.84, 19.9) mm, rotated rx 180 ry 0 rz -180 deg; joints [1.893, 67.23, -30.46, 3.16, -36.811, -2.531]
  Call Extruder 0.01786
  MoveL (T19259) to (112.56, 103.84, 19.9) mm, rotated rx 180 ry 0 rz -180 deg; joints [1.893, 67.23, -30.46, 3.16, -36.811, -2.531]
  Call Extruder 0.0573
  MoveL (T19260) to (113.88, 105.16, 19.9) mm, rotated rx 180 ry 0 rz -180 deg; joints [1.893, 67.23, -30.46, 3.16, -36.811, -2.531]
  Call Extruder 0.01786
  MoveL (T19261) to (113.3, 105.16, 19.9) mm, rotated rx 180 ry 0 rz -180 deg; joints [1.893, 67.23, -30.46, 3.16, -36.811, -2.531]
  Call Extruder 0.0573
  MoveL (T19262) to (111.98, 103.84, 19.9) mm, rotated rx 180 ry 0 rz -180 deg; joints [1.895, 67.093, -30.203, 3.155, -36.931, -2.523]
  Call Extruder 0.01786
  MoveL (T19263) to (111.4, 103.84, 19.9) mm, rotated rx 180 ry 0 rz -180 deg; joints [1.895, 67.093, -30.203, 3.155, -36.931, -2.523]
  Call Extruder 0.0573
  MoveL (T19264) to (112.72, 105.16, 19.9) mm, rotated rx 180 ry 0 rz -180 deg; joints [2.319, 66.136, -28.409, 3.787, -37.788, -2.994]
  Call Extruder 0.01786
  MoveL (T19265) to (112.13, 105.16, 19.9) mm, rotated rx 180 ry 0 rz -180 deg; joints [2.319, 66.136, -28.409, 3.787, -37.788, -2.994]
  Call Extruder 0.0573
  MoveL (T19266) to (110.81, 103.84, 19.9) mm, rotated rx 180 ry 0 rz -180 deg; joints [2.44, 66.148, -28.431, 3.984, -37.784, -3.151]
  Call Extruder 0.01786
  MoveL (T19267) to (110.23, 103.84, 19.9) mm, rotated rx 180 ry 0 rz -180 deg; joints [2.44, 66.148, -28.431, 3.984, -37.784, -3.151]
  Call Extruder 0.0573
  MoveL (T19268) to (111.55, 105.16, 19.9) mm, rotated rx 180 ry 0 rz -180 deg; joints [3.266, 68.429, -32.712, 5.583, -35.846, -4.531]
  Call Extruder 0.01786
  MoveL (T19269) to (110.97, 105.16, 19.9) mm, rotated rx 180 ry 0 rz -180 deg; joints [3.266, 68.429, -32.712, 5.583, -35.846, -4.531]
  Call Extruder 0.0573
  MoveL (T19270) to (109.65, 103.84, 19.9) mm, rotated rx 180 ry 0 rz -180 deg; joints [3.266, 68.429, -32.712, 5.583, -35.846, -4.531]
  Call Extruder 0.01786
  MoveL (T19271) to (109.07, 103.84, 19.9) mm, rotated rx 180 ry 0 rz -180 deg; joints [3.26, 68.742, -33.301, 5.609, -35.572, -4.567]
  Call Extruder 0.0573
  MoveL (T19272) to (110.39, 105.16, 19.9) mm, rotated rx 180 ry 0 rz -180 deg; joints [3.26, 68.742, -33.301, 5.609, -35.572, -4.567]
  Call Extruder 0.01786
  MoveL (T19273) to (109.81, 105.16, 19.9) mm, rotated rx 180 ry 0 rz -180 deg; joints [2.685, 70.174, -35.99, 4.771, -34.277, -3.945]
  Call Extruder 0.0573
  MoveL (T19274) to (108.49, 103.84, 19.9) mm, rotated rx 180 ry 0 rz -180 deg; joints [2.685, 70.174, -35.99, 4.771, -34.277, -3.945]
  Call Extruder 0.01786
  MoveL (T19275) to (107.91, 103.84, 19.9) mm, rotated rx 180 ry 0 rz -180 deg; joints [2.685, 70.174, -35.99, 4.771, -34.277, -3.945]
  Call Extruder 0.0573
  MoveL (T19276) to (109.23, 105.16, 19.9) mm, rotated rx 180 ry 0 rz -180 deg; joints [2.685, 70.174, -35.99, 4.771, -34.277, -3.945]
  Call Extruder 0.01786
  MoveL (T19277) to (108.65, 105.16, 19.9) mm, rotated rx 180 ry 0 rz -180 deg; joints [2.754, 70.394, -36.402, 4.918, -34.089, -4.076]
  Call Extruder 0.0573
  MoveL (T19278) to (107.33, 103.84, 19.9) mm, rotated rx 180 ry 0 rz -180 deg; joints [2.762, 70.456, -36.52, 4.939, -34.035, -4.096]
  Call Extruder 0.01786
  MoveL (T19279) to (106.75, 103.84, 19.9) mm, rotated rx 180 ry 0 rz -180 deg; joints [2.762, 70.456, -36.52, 4.939, -34.035, -4.096]
  Call Extruder 0.0573
  MoveL (T19280) to (108.07, 105.16, 19.9) mm, rotated rx 180 ry 0 rz -180 deg; joints [2.762, 70.456, -36.52, 4.939, -34.035, -4.096]
  Call Extruder 0.01786
  MoveL (T19281) to (107.49, 105.16, 19.9) mm, rotated rx 180 ry 0 rz -180 deg; joints [2.756, 70.84, -37.241, 4.971, -33.699, -4.139]
  Call Extruder 0.0573
  MoveL (T19282) to (106.17, 103.84, 19.9) mm, rotated rx 180 ry 0 rz -180 deg; joints [2.756, 70.84, -37.241, 4.971, -33.699, -4.139]
  Call Extruder 0.01786
  MoveL (T19283) to (105.59, 103.84, 19.9) mm, rotated rx 180 ry 0 rz -180 deg; joints [2.633, 71.13, -37.785, 4.782, -33.436, -3.994]
  Call Extruder 0.08219
  MoveL (T19284) to (107.48, 105.73, 19.9) mm, rotated rx 180 ry 0 rz -180 deg; joints [2.633, 71.13, -37.785, 4.782, -33.436, -3.994]
  Call Extruder 0.01786
  MoveL (T19285) to (107.48, 106.32, 19.9) mm, rotated rx 180 ry 0 rz -180 deg; joints [2.633, 71.13, -37.785, 4.782, -33.436, -3.994]
  Call Extruder 0.10744
  MoveL (T19286) to (105.01, 103.84, 19.9) mm, rotated rx 180 ry 0 rz -180 deg; joints [2.633, 71.13, -37.785, 4.782, -33.436, -3.994]
  Call Extruder 0.01786
  MoveL (T19287) to (104.42, 103.84, 19.9) mm, rotated rx 180 ry 0 rz -180 deg; joints [2.712, 70.916, -37.383, 4.9, -33.629, -4.083]
  Call Extruder 0.1327
  MoveL (T19288) to (107.48, 106.9, 19.9) mm, rotated rx 180 ry 0 rz -180 deg; joints [2.712, 70.916, -37.383, 4.9, -33.629, -4.083]
  Call Extruder 0.01087
  MoveL (T19289) to (107.48, 107.25, 19.9) mm, rotated rx 180 ry 0 rz -180 deg; joints [2.714, 70.736, -37.046, 4.885, -33.787, -4.063]
  Call Extruder 0.01602
  MoveL (T19290) to (107.72, 107.72, 19.9) mm, rotated rx 180 ry 0 rz -180 deg; joints [2.714, 70.736, -37.046, 4.885, -33.787, -4.063]
  Call Extruder 0.16825
  MoveL (T19291) to (103.84, 103.84, 19.9) mm, rotated rx 180 ry 0 rz -180 deg; joints [2.592, 71.067, -37.667, 4.702, -33.489, -3.924]
  Call Extruder 0.01786
  MoveL (T19292) to (103.84, 104.42, 19.9) mm, rotated rx 180 ry 0 rz -180 deg; joints [2.592, 71.067, -37.667, 4.702, -33.489, -3.924]
  Call Extruder 0.19454
  MoveL (T19293) to (108.32, 108.9, 19.9) mm, rotated rx 180 ry 0 rz -180 deg; joints [2.592, 71.067, -37.667, 4.702, -33.489, -3.924]
  Call Extruder 0.04092
  MoveL (T19294) to (108.92, 110.09, 19.9) mm, rotated rx 180 ry 0 rz -180 deg; joints [2.532, 71.059, -37.651, 4.591, -33.492, -3.832]
  Call Extruder 0.22084
  MoveL (T19295) to (103.84, 105.01, 19.9) mm, rotated rx 180 ry 0 rz -180 deg; joints [2.532, 71.059, -37.651, 4.591, -33.492, -3.832]
  Call Extruder 0.01786
  MoveL (T19296) to (103.84, 105.59, 19.9) mm, rotated rx 180 ry 0 rz -180 deg; joints [2.532, 71.059, -37.651, 4.591, -33.492, -3.832]
  Call Extruder 0.24714
  MoveL (T19297) to (109.53, 111.27, 19.9) mm, rotated rx 180 ry 0 rz -180 deg; joints [2.717, 70.558, -36.711, 4.871, -33.943, -4.044]
  Call Extruder 0.04092
  MoveL (T19298) to (110.13, 112.46, 19.9) mm, rotated rx 180 ry 0 rz -180 deg; joints [2.719, 70.475, -36.555, 4.864, -34.016, -4.034]
  Call Extruder 0.27344
  MoveL (T19299) to (103.84, 106.17, 19.9) mm, rotated rx 180 ry 0 rz -180 deg; joints [2.719, 70.475, -36.555, 4.864, -34.016, -4.034]
  Call Extruder 0.01786
  MoveL (T19300) to (103.84, 106.75, 19.9) mm, rotated rx 180 ry 0 rz -180 deg; joints [2.719, 70.475, -36.555, 4.864, -34.016, -4.034]
  Call Extruder 0.29974
  MoveL (T19301) to (110.74, 113.64, 19.9) mm, rotated rx 180 ry 0 rz -180 deg; joints [2.717, 70.459, -36.525, 4.858, -34.029, -4.029]
  Call Extruder 0.04092
  MoveL (T19302) to (111.34, 114.83, 19.9) mm, rotated rx 180 ry 0 rz -180 deg; joints [2.717, 70.459, -36.525, 4.858, -34.029, -4.029]
  Call Extruder 0.32604
  MoveL (T19303) to (103.84, 107.33, 19.9) mm, rotated rx 180 ry 0 rz -180 deg; joints [2.717, 70.459, -36.525, 4.858, -34.029, -4.029]
  Call Extruder 0.01786
  MoveL (T19304) to (103.84, 107.91, 19.9) mm, rotated rx 180 ry 0 rz -180 deg; joints [2.717, 70.459, -36.525, 4.858, -34.029, -4.029]
  Call Extruder 0.34996
  MoveL (T19305) to (111.89, 115.96, 19.9) mm, rotated rx 180 ry 0 rz -180 deg; joints [2.705, 70.421, -36.454, 4.833, -34.062, -4.007]
  Call Extruder 0.01786
  MoveL (T19306) to (111.31, 115.96, 19.9) mm, rotated rx 180 ry 0 rz -180 deg; joints [2.705, 70.421, -36.454, 4.833, -34.062, -4.007]
  Call Extruder 0.32471
  MoveL (T19307) to (103.84, 108.49, 19.9) mm, rotated rx 180 ry 0 rz -180 deg; joints [2.705, 70.421, -36.454, 4.833, -34.062, -4.007]
  Call Extruder 0.01786
  MoveL (T19308) to (103.84, 109.07, 19.9) mm, rotated rx 180 ry 0 rz -180 deg; joints [2.705, 70.421, -36.454, 4.833, -34.062, -4.007]
  Call Extruder 0.29945
  MoveL (T19309) to (110.73, 115.96, 19.9) mm, rotated rx 180 ry 0 rz -180 deg; joints [2.471, 71.051, -37.636, 4.481, -33.495, -3.739]
  Call Extruder 0.01786
  MoveL (T19310) to (110.15, 115.96, 19.9) mm, rotated rx 180 ry 0 rz -180 deg; joints [2.471, 71.051, -37.636, 4.481, -33.495, -3.739]
  Call Extruder 0.2742
  MoveL (T19311) to (103.84, 109.65, 19.9) mm, rotated rx 180 ry 0 rz -180 deg; joints [2.41, 71.043, -37.622, 4.37, -33.498, -3.646]
  Call Extruder 0.01786
  MoveL (T19312) to (103.84, 110.23, 19.9) mm, rotated rx 180 ry 0 rz -180 deg; joints [2.41, 71.043, -37.622, 4.37, -33.498, -3.646]
  Call Extruder 0.24895
  MoveL (T19313) to (109.57, 115.96, 19.9) mm, rotated rx 180 ry 0 rz -180 deg; joints [2.41, 71.043, -37.622, 4.37, -33.498, -3.646]
  Call Extruder 0.01786
  MoveL (T19314) to (108.99, 115.96, 19.9) mm, rotated rx 180 ry 0 rz -180 deg; joints [2.676, 70.329, -36.281, 4.772, -34.14, -3.952]
  Call Extruder 0.22369
  MoveL (T19315) to (103.84, 110.82, 19.9) mm, rotated rx 180 ry 0 rz -180 deg; joints [2.676, 70.329, -36.281, 4.772, -34.14, -3.952]
  Call Extruder 0.01786
  MoveL (T19316) to (103.84, 111.4, 19.9) mm, rotated rx 180 ry 0 rz -180 deg; joints [2.676, 70.329, -36.281, 4.772, -34.14, -3.952]
  Call Extruder 0.19844
  MoveL (T19317) to (108.41, 115.96, 19.9) mm, rotated rx 180 ry 0 rz -180 deg; joints [2.647, 70.238, -36.109, 4.71, -34.218, -3.898]
  Call Extruder 0.01786
  MoveL (T19318) to (107.83, 115.96, 19.9) mm, rotated rx 180 ry 0 rz -180 deg; joints [2.647, 70.238, -36.109, 4.71, -34.218, -3.898]
  Call Extruder 0.17318
  MoveL (T19319) to (103.84, 111.98, 19.9) mm, rotated rx 180 ry 0 rz -180 deg; joints [2.647, 70.238, -36.109, 4.71, -34.218, -3.898]
  Call Extruder 0.01786
  MoveL (T19320) to (103.84, 112.56, 19.9) mm, rotated rx 180 ry 0 rz -180 deg; joints [2.35, 71.035, -37.608, 4.26, -33.5, -3.554]
  Call Extruder 0.1616
  MoveL (T19321) to (107.56, 116.28, 19.9) mm, rotated rx 180 ry 0 rz -180 deg; joints [2.35, 71.035, -37.608, 4.26, -33.5, -3.554]
  Call Extruder 0.01786
  MoveL (T19322) to (107.56, 116.86, 19.9) mm, rotated rx 180 ry 0 rz -180 deg; joints [2.289, 71.028, -37.594, 4.149, -33.503, -3.462]
  Call Extruder 0.1616
  MoveL (T19323) to (103.84, 113.14, 19.9) mm, rotated rx 180 ry 0 rz -180 deg; joints [2.289, 71.028, -37.594, 4.149, -33.503, -3.462]
  Call Extruder 0.01786
  MoveL (T19324) to (103.84, 113.72, 19.9) mm, rotated rx 180 ry 0 rz -180 deg; joints [2.618, 70.146, -35.937, 4.649, -34.297, -3.843]
  Call Extruder 0.1616
  MoveL (T19325) to (107.56, 117.44, 19.9) mm, rotated rx 180 ry 0 rz -180 deg; joints [2.618, 70.146, -35.937, 4.649, -34.297, -3.843]
  Call Extruder 0.01786
  MoveL (T19326) to (107.56, 118.02, 19.9) mm, rotated rx 180 ry 0 rz -180 deg; joints [2.618, 70.146, -35.937, 4.649, -34.297, -3.843]
  Call Extruder 0.1616
  MoveL (T19327) to (103.84, 114.3, 19.9) mm, rotated rx 180 ry 0 rz -180 deg; joints [2.588, 70.055, -35.767, 4.588, -34.374, -3.789]
  Call Extruder 0.01786
  MoveL (T19328) to (103.84, 114.88, 19.9) mm, rotated rx 180 ry 0 rz -180 deg; joints [2.588, 70.055, -35.767, 4.588, -34.374, -3.789]
  Call Extruder 0.1616
  MoveL (T19329) to (107.56, 118.6, 19.9) mm, rotated rx 180 ry 0 rz -180 deg; joints [2.228, 71.021, -37.581, 4.039, -33.506, -3.369]
  Call Extruder 0.01786
  MoveL (T19330) to (107.56, 119.18, 19.9) mm, rotated rx 180 ry 0 rz -180 deg; joints [2.228, 71.021, -37.581, 4.039, -33.506, -3.369]
  Call Extruder 0.16957
  MoveL (T19331) to (103.66, 115.28, 19.9) mm, rotated rx 180 ry 0 rz -180 deg; joints [2.228, 71.021, -37.581, 4.039, -33.506, -3.369]
  Set speed (45.0 mm/s)
  Call Extruder -1.6
  MoveL (T19332) to (103.66, 115.28, 19.9) mm, rotated rx 180 ry 0 rz -180 deg; joints [2.168, 71.014, -37.567, 3.928, -33.508, -3.277]
  Set speed (120.0 mm/s)
  MoveL (T19333) to (103.66, 115.28, 19.9) mm, rotated rx 180 ry 0 rz -180 deg; joints [2.168, 71.014, -37.567, 3.928, -33.508, -3.277]
  Call Extruder -0.38
  MoveL (T19334) to (104.42, 116.03, 19.9) mm, rotated rx 180 ry 0 rz -180 deg; joints [2.559, 69.965, -35.597, 4.527, -34.452, -3.736]
  Set speed (45.0 mm/s)
  Call Extruder -0.02
  MoveL (T19335) to (104.42, 116.03, 19.9) mm, rotated rx 180 ry 0 rz -180 deg; joints [2.559, 69.965, -35.597, 4.527, -34.452, -3.736]
  Set speed (150.0 mm/s)
  MoveL (T19336) to (104.42, 116.03, 21.9) mm, rotated rx 180 ry 0 rz -180 deg; joints [2.559, 69.965, -35.597, 4.527, -34.452, -3.736]
  MoveL (T19337) to (117.77, 105.57, 21.9) mm, rotated rx 180 ry 0 rz -180 deg; joints [2.53, 69.874, -35.427, 4.467, -34.529, -3.682]
  MoveL (T19338) to (117.77, 105.57, 19.9) mm, rotated rx 180 ry 0 rz -180 deg; joints [2.53, 69.874, -35.427, 4.467, -34.529, -3.682]
  Set speed (40.0 mm/s)
  Call Extruder 2.0
  MoveL (T19339) to (117.77, 105.57, 19.9) mm, rotated rx 180 ry 0 rz -180 deg; joints [2.53, 69.874, -35.427, 4.467, -34.529, -3.682]
  Call Extruder 0.14703
  MoveL (T19340) to (121.16, 108.96, 19.9) mm, rotated rx 180 ry 0 rz -180 deg; joints [2.53, 69.874, -35.427, 4.467, -34.529, -3.682]
  Call Extruder 0.01786
  MoveL (T19341) to (121.16, 109.54, 19.9) mm, rotated rx 180 ry 0 rz -180 deg; joints [2.107, 71.007, -37.555, 3.818, -33.511, -3.185]
  Call Extruder 0.13907
  MoveL (T19342) to (117.96, 106.34, 19.9) mm, rotated rx 180 ry 0 rz -180 deg; joints [2.107, 71.007, -37.555, 3.818, -33.511, -3.185]
  Call Extruder 0.01786
  MoveL (T19343) to (117.96, 106.92, 19.9) mm, rotated rx 180 ry 0 rz -180 deg; joints [2.107, 71.007, -37.555, 3.818, -33.511, -3.185]
  Call Extruder 0.13907
  MoveL (T19344) to (121.16, 110.12, 19.9) mm, rotated rx 180 ry 0 rz -180 deg; joints [2.046, 71.001, -37.542, 3.708, -33.513, -3.092]
  Call Extruder 0.01786
  MoveL (T19345) to (121.16, 110.7, 19.9) mm, rotated rx 180 ry 0 rz -180 deg; joints [2.046, 71.001, -37.542, 3.708, -33.513, -3.092]
  Call Extruder 0.13907
  MoveL (T19346) to (117.96, 107.5, 19.9) mm, rotated rx 180 ry 0 rz -180 deg; joints [2.046, 71.001, -37.542, 3.708, -33.513, -3.092]
  Call Extruder 0.01786
  MoveL (T19347) to (117.96, 108.08, 19.9) mm, rotated rx 180 ry 0 rz -180 deg; joints [2.479, 69.842, -35.366, 4.373, -34.554, -3.604]
  Call Extruder 0.13907
  MoveL (T19348) to (121.16, 111.28, 19.9) mm, rotated rx 180 ry 0 rz -180 deg; joints [2.479, 69.842, -35.366, 4.373, -34.554, -3.604]
  Call Extruder 0.01786
  MoveL (T19349) to (121.16, 111.86, 19.9) mm, rotated rx 180 ry 0 rz -180 deg; joints [2.418, 69.835, -35.353, 4.265, -34.556, -3.514]
  Call Extruder 0.13907
  MoveL (T19350) to (117.96, 108.66, 19.9) mm, rotated rx 180 ry 0 rz -180 deg; joints [1.985, 70.994, -37.53, 3.597, -33.516, -3]
  Call Extruder 0.01786
  MoveL (T19351) to (117.96, 109.24, 19.9) mm, rotated rx 180 ry 0 rz -180 deg; joints [1.985, 70.994, -37.53, 3.597, -33.516, -3]
  Call Extruder 0.13907
  MoveL (T19352) to (121.16, 112.44, 19.9) mm, rotated rx 180 ry 0 rz -180 deg; joints [1.925, 70.988, -37.519, 3.487, -33.518, -2.908]
  Call Extruder 0.01786
  MoveL (T19353) to (121.16, 113.02, 19.9) mm, rotated rx 180 ry 0 rz -180 deg; joints [1.925, 70.988, -37.519, 3.487, -33.518, -2.908]
  Call Extruder 0.15905
  MoveL (T19354) to (117.5, 109.36, 19.9) mm, rotated rx 180 ry 0 rz -180 deg; joints [1.925, 70.988, -37.519, 3.487, -33.518, -2.908]
  Call Extruder 0.01786
  MoveL (T19355) to (116.92, 109.36, 19.9) mm, rotated rx 180 ry 0 rz -180 deg; joints [2.356, 69.828, -35.339, 4.156, -34.559, -3.425]
  Call Extruder 0.1843
  MoveL (T19356) to (121.16, 113.6, 19.9) mm, rotated rx 180 ry 0 rz -180 deg; joints [2.356, 69.828, -35.339, 4.156, -34.559, -3.425]
  Call Extruder 0.01786
  MoveL (T19357) to (121.16, 114.19, 19.9) mm, rotated rx 180 ry 0 rz -180 deg; joints [2.295, 69.821, -35.326, 4.048, -34.562, -3.336]
  Call Extruder 0.20956
  MoveL (T19358) to (116.33, 109.36, 19.9) mm, rotated rx 180 ry 0 rz -180 deg; joints [2.295, 69.821, -35.326, 4.048, -34.562, -3.336]
  Call Extruder 0.01786
  MoveL (T19359) to (115.75, 109.36, 19.9) mm, rotated rx 180 ry 0 rz -180 deg; joints [2.295, 69.821, -35.326, 4.048, -34.562, -3.336]
  Call Extruder 0.23481
  MoveL (T19360) to (121.16, 114.77, 19.9) mm, rotated rx 180 ry 0 rz -180 deg; joints [1.864, 70.982, -37.508, 3.377, -33.52, -2.816]
  Call Extruder 0.01786
  MoveL (T19361) to (121.16, 115.35, 19.9) mm, rotated rx 180 ry 0 rz -180 deg; joints [1.864, 70.982, -37.508, 3.377, -33.52, -2.816]
  Call Extruder 0.26007
  MoveL (T19362) to (115.17, 109.36, 19.9) mm, rotated rx 180 ry 0 rz -180 deg; joints [1.83, 70.979, -37.501, 3.314, -33.522, -2.764]
  Call Extruder 0.01786
  MoveL (T19363) to (114.59, 109.36, 19.9) mm, rotated rx 180 ry 0 rz -180 deg; joints [1.83, 70.979, -37.501, 3.314, -33.522, -2.764]
  Call Extruder 0.28532
  MoveL (T19364) to (121.16, 115.93, 19.9) mm, rotated rx 180 ry 0 rz -180 deg; joints [1.83, 70.9, -37.353, 3.31, -33.591, -2.758]
  Call Extruder 0.01786
  MoveL (T19365) to (121.16, 116.51, 19.9) mm, rotated rx 180 ry 0 rz -180 deg; joints [1.83, 70.9, -37.353, 3.31, -33.591, -2.758]
  Call Extruder 0.31058
  MoveL (T19366) to (114.01, 109.36, 19.9) mm, rotated rx 180 ry 0 rz -180 deg; joints [2.234, 69.814, -35.313, 3.94, -34.564, -3.246]
  Call Extruder 0.01786
  MoveL (T19367) to (113.43, 109.36, 19.9) mm, rotated rx 180 ry 0 rz -180 deg; joints [2.234, 69.814, -35.313, 3.94, -34.564, -3.246]
  Call Extruder 0.33583
  MoveL (T19368) to (121.16, 117.09, 19.9) mm, rotated rx 180 ry 0 rz -180 deg; joints [2.173, 69.808, -35.301, 3.832, -34.566, -3.157]
  Call Extruder 0.01786
  MoveL (T19369) to (121.16, 117.67, 19.9) mm, rotated rx 180 ry 0 rz -180 deg; joints [2.173, 69.808, -35.301, 3.832, -34.566, -3.157]
  Call Extruder 0.31968
  MoveL (T19370) to (113.8, 110.32, 19.9) mm, rotated rx 180 ry 0 rz -180 deg; joints [2.173, 69.808, -35.301, 3.832, -34.566, -3.157]
  Call Extruder 0.04109
  MoveL (T19371) to (114.41, 111.51, 19.9) mm, rotated rx 180 ry 0 rz -180 deg; joints [1.832, 70.72, -37.016, 3.3, -33.748, -2.745]
  Call Extruder 0.29321
  MoveL (T19372) to (121.16, 118.25, 19.9) mm, rotated rx 180 ry 0 rz -180 deg; joints [1.832, 70.72, -37.016, 3.3, -33.748, -2.745]
  Call Extruder 0.01786
  MoveL (T19373) to (121.16, 118.83, 19.9) mm, rotated rx 180 ry 0 rz -180 deg; joints [1.832, 70.72, -37.016, 3.3, -33.748, -2.745]
  Call Extruder 0.26675
  MoveL (T19374) to (115.02, 112.7, 19.9) mm, rotated rx 180 ry 0 rz -180 deg; joints [1.832, 70.72, -37.016, 3.3, -33.748, -2.745]
  Call Extruder 0.04109
  MoveL (T19375) to (115.63, 113.89, 19.9) mm, rotated rx 180 ry 0 rz -180 deg; joints [1.832, 70.72, -37.016, 3.3, -33.748, -2.745]
  Call Extruder 0.24028
  MoveL (T19376) to (121.16, 119.41, 19.9) mm, rotated rx 180 ry 0 rz -180 deg; joints [1.834, 70.542, -36.681, 3.29, -33.905, -2.731]
  Call Extruder 0.01786
  MoveL (T19377) to (121.16, 119.99, 19.9) mm, rotated rx 180 ry 0 rz -180 deg; joints [1.834, 70.542, -36.681, 3.29, -33.905, -2.731]
  Call Extruder 0.21381
  MoveL (T19378) to (116.24, 115.08, 19.9) mm, rotated rx 180 ry 0 rz -180 deg; joints [1.834, 70.542, -36.681, 3.29, -33.905, -2.731]
  Call Extruder 0.04109
  MoveL (T19379) to (116.85, 116.27, 19.9) mm, rotated rx 180 ry 0 rz -180 deg; joints [1.834, 70.542, -36.681, 3.29, -33.905, -2.731]
  Call Extruder 0.18734
  MoveL (T19380) to (121.16, 120.58, 19.9) mm, rotated rx 180 ry 0 rz -180 deg; joints [2.112, 69.801, -35.289, 3.724, -34.568, -3.068]
  Call Extruder 0.01786
  MoveL (T19381) to (121.16, 121.16, 19.9) mm, rotated rx 180 ry 0 rz -180 deg; joints [2.112, 69.801, -35.289, 3.724, -34.568, -3.068]
  Call Extruder 0.16087
  MoveL (T19382) to (117.45, 117.45, 19.9) mm, rotated rx 180 ry 0 rz -180 deg; joints [2.112, 69.801, -35.289, 3.724, -34.568, -3.068]
  Call Extruder 0.02137
  MoveL (T19383) to (117.77, 118.07, 19.9) mm, rotated rx 180 ry 0 rz -180 deg; joints [2.053, 69.795, -35.278, 3.621, -34.571, -2.983]
  Call Extruder 0.00857
  MoveL (T19384) to (117.77, 118.35, 19.9) mm, rotated rx 180 ry 0 rz -180 deg; joints [2.053, 69.795, -35.278, 3.621, -34.571, -2.983]
  Call Extruder 0.12185
  MoveL (T19385) to (120.58, 121.16, 19.9) mm, rotated rx 180 ry 0 rz -180 deg; joints [2.048, 69.801, -35.288, 3.612, -34.566, -2.976]
  Call Extruder 0.01786
  MoveL (T19386) to (119.99, 121.16, 19.9) mm, rotated rx 180 ry 0 rz -180 deg; joints [2.048, 69.801, -35.288, 3.612, -34.566, -2.976]
  Call Extruder 0.09659
  MoveL (T19387) to (117.77, 118.93, 19.9) mm, rotated rx 180 ry 0 rz -180 deg; joints [2.048, 69.801, -35.288, 3.612, -34.566, -2.976]
  Call Extruder 0.01786
  MoveL (T19388) to (117.77, 119.52, 19.9) mm, rotated rx 180 ry 0 rz -180 deg; joints [1.816, 70.419, -36.451, 3.248, -34.011, -2.694]
  Call Extruder 0.07134
  MoveL (T19389) to (119.41, 121.16, 19.9) mm, rotated rx 180 ry 0 rz -180 deg; joints [1.816, 70.419, -36.451, 3.248, -34.011, -2.694]
  Call Extruder 0.01786
  MoveL (T19390) to (118.83, 121.16, 19.9) mm, rotated rx 180 ry 0 rz -180 deg; joints [1.835, 69.993, -35.65, 3.251, -34.386, -2.684]
  Call Extruder 0.04608
  MoveL (T19391) to (117.77, 120.1, 19.9) mm, rotated rx 180 ry 0 rz -180 deg; joints [1.835, 69.993, -35.65, 3.251, -34.386, -2.684]
  Call Extruder 0.00206
  MoveL (T19392) to (117.77, 120.16, 19.9) mm, rotated rx 180 ry 0 rz -180 deg; joints [1.835, 69.993, -35.65, 3.251, -34.386, -2.684]
  Call Extruder 0.0158
  MoveL (T19393) to (117.26, 120.16, 19.9) mm, rotated rx 180 ry 0 rz -180 deg; joints [1.835, 69.993, -35.65, 3.251, -34.386, -2.684]
  Call Extruder 0.04317
  MoveL (T19394) to (118.25, 121.16, 19.9) mm, rotated rx 180 ry 0 rz -180 deg; joints [1.835, 69.993, -35.65, 3.251, -34.386, -2.684]
  Call Extruder 0.01786
  MoveL (T19395) to (117.67, 121.16, 19.9) mm, rotated rx 180 ry 0 rz -180 deg; joints [1.835, 69.993, -35.65, 3.251, -34.386, -2.684]
  Call Extruder 0.04317
  MoveL (T19396) to (116.68, 120.16, 19.9) mm, rotated rx 180 ry 0 rz -180 deg; joints [1.835, 69.993, -35.65, 3.251, -34.386, -2.684]
  Call Extruder 0.01786
  MoveL (T19397) to (116.1, 120.16, 19.9) mm, rotated rx 180 ry 0 rz -180 deg; joints [1.603, 70.624, -36.834, 2.881, -33.823, -2.394]
  Call Extruder 0.04317
  MoveL (T19398) to (117.09, 121.16, 19.9) mm, rotated rx 180 ry 0 rz -180 deg; joints [1.603, 70.624, -36.834, 2.881, -33.823, -2.394]
  Call Extruder 0.01786
  MoveL (T19399) to (116.51, 121.16, 19.9) mm, rotated rx 180 ry 0 rz -180 deg; joints [1.599, 70.628, -36.842, 2.874, -33.819, -2.389]
  Call Extruder 0.04317
  MoveL (T19400) to (115.52, 120.16, 19.9) mm, rotated rx 180 ry 0 rz -180 deg; joints [1.599, 70.628, -36.842, 2.874, -33.819, -2.389]
  Call Extruder 0.01786
  MoveL (T19401) to (114.93, 120.16, 19.9) mm, rotated rx 180 ry 0 rz -180 deg; joints [1.599, 70.628, -36.842, 2.874, -33.819, -2.389]
  Call Extruder 0.04317
  MoveL (T19402) to (115.93, 121.16, 19.9) mm, rotated rx 180 ry 0 rz -180 deg; joints [1.539, 70.623, -36.833, 2.766, -33.821, -2.298]
  Call Extruder 0.01786
  MoveL (T19403) to (115.35, 121.16, 19.9) mm, rotated rx 180 ry 0 rz -180 deg; joints [1.539, 70.623, -36.833, 2.766, -33.821, -2.298]
  Call Extruder 0.04317
  MoveL (T19404) to (114.35, 120.16, 19.9) mm, rotated rx 180 ry 0 rz -180 deg; joints [1.817, 69.869, -35.417, 3.21, -34.494, -2.647]
  Call Extruder 0.01786
  MoveL (T19405) to (113.77, 120.16, 19.9) mm, rotated rx 180 ry 0 rz -180 deg; joints [1.817, 69.869, -35.417, 3.21, -34.494, -2.647]
  Call Extruder 0.04317
  MoveL (T19406) to (114.77, 121.16, 19.9) mm, rotated rx 180 ry 0 rz -180 deg; joints [1.817, 69.869, -35.417, 3.21, -34.494, -2.647]
  Call Extruder 0.01786
  MoveL (T19407) to (114.18, 121.16, 19.9) mm, rotated rx 180 ry 0 rz -180 deg; joints [1.819, 69.693, -35.087, 3.201, -34.648, -2.634]
  Call Extruder 0.04317
  MoveL (T19408) to (113.19, 120.16, 19.9) mm, rotated rx 180 ry 0 rz -180 deg; joints [1.819, 69.693, -35.087, 3.201, -34.648, -2.634]
  Call Extruder 0.01786
  MoveL (T19409) to (112.61, 120.16, 19.9) mm, rotated rx 180 ry 0 rz -180 deg; joints [1.819, 69.693, -35.087, 3.201, -34.648, -2.634]
  Call Extruder 0.04317
  MoveL (T19410) to (113.6, 121.16, 19.9) mm, rotated rx 180 ry 0 rz -180 deg; joints [1.477, 70.618, -36.824, 2.653, -33.823, -2.205]
  Call Extruder 0.01786
  MoveL (T19411) to (113.02, 121.16, 19.9) mm, rotated rx 180 ry 0 rz -180 deg; joints [1.477, 70.618, -36.824, 2.653, -33.823, -2.205]
  Call Extruder 0.04317
  MoveL (T19412) to (112.03, 120.16, 19.9) mm, rotated rx 180 ry 0 rz -180 deg; joints [1.477, 70.618, -36.824, 2.653, -33.823, -2.205]
  Call Extruder 0.01786
  MoveL (T19413) to (111.45, 120.16, 19.9) mm, rotated rx 180 ry 0 rz -180 deg; joints [1.414, 70.614, -36.816, 2.541, -33.824, -2.111]
  Call Extruder 0.04317
  MoveL (T19414) to (112.44, 121.16, 19.9) mm, rotated rx 180 ry 0 rz -180 deg; joints [1.414, 70.614, -36.816, 2.541, -33.824, -2.111]
  Call Extruder 0.01786
  MoveL (T19415) to (111.86, 121.16, 19.9) mm, rotated rx 180 ry 0 rz -180 deg; joints [1.414, 70.614, -36.816, 2.541, -33.824, -2.111]
  Call Extruder 0.04317
  MoveL (T19416) to (110.87, 120.16, 19.9) mm, rotated rx 180 ry 0 rz -180 deg; joints [1.414, 70.614, -36.816, 2.541, -33.824, -2.111]
  Call Extruder 0.01786
  MoveL (T19417) to (110.29, 120.16, 19.9) mm, rotated rx 180 ry 0 rz -180 deg; joints [1.821, 69.518, -34.758, 3.192, -34.802, -2.622]
  Call Extruder 0.04317
  MoveL (T19418) to (111.28, 121.16, 19.9) mm, rotated rx 180 ry 0 rz -180 deg; joints [1.821, 69.518, -34.758, 3.192, -34.802, -2.622]
  Call Extruder 0.01786
  MoveL (T19419) to (110.7, 121.16, 19.9) mm, rotated rx 180 ry 0 rz -180 deg; joints [1.821, 69.518, -34.758, 3.192, -34.802, -2.622]
  Call Extruder 0.04317
  MoveL (T19420) to (109.71, 120.16, 19.9) mm, rotated rx 180 ry 0 rz -180 deg; joints [1.823, 69.345, -34.432, 3.184, -34.954, -2.61]
  Call Extruder 0.01786
  MoveL (T19421) to (109.12, 120.16, 19.9) mm, rotated rx 180 ry 0 rz -180 deg; joints [1.823, 69.345, -34.432, 3.184, -34.954, -2.61]
  Call Extruder 0.04317
  MoveL (T19422) to (110.12, 121.16, 19.9) mm, rotated rx 180 ry 0 rz -180 deg; joints [1.823, 69.345, -34.432, 3.184, -34.954, -2.61]
  Call Extruder 0.01786
  MoveL (T19423) to (109.54, 121.16, 19.9) mm, rotated rx 180 ry 0 rz -180 deg; joints [1.4, 70.476, -36.556, 2.507, -33.945, -2.081]
  Call Extruder 0.05113
  MoveL (T19424) to (108.36, 119.98, 19.9) mm, rotated rx 180 ry 0 rz -180 deg; joints [1.4, 70.476, -36.556, 2.507, -33.945, -2.081]
  Set speed (150.0 mm/s)
  MoveL (T19425) to (109.14, 121.34, 19.9) mm, rotated rx 180 ry 0 rz -180 deg; joints [1.4, 70.476, -36.556, 2.507, -33.945, -2.081]
  Set speed (40.0 mm/s)
  MoveL (T19426) to (109.14, 121.34, 19.9) mm, rotated rx 180 ry 0 rz -180 deg; joints [1.401, 70.295, -36.216, 2.5, -34.104, -2.07]
  Call Extruder 0.05113
  MoveL (T19427) to (107.96, 120.16, 19.9) mm, rotated rx 180 ry 0 rz -180 deg; joints [1.401, 70.295, -36.216, 2.5, -34.104, -2.07]
  Call Extruder 0.01234
  MoveL (T19428) to (107.56, 120.16, 19.9) mm, rotated rx 180 ry 0 rz -180 deg; joints [1.401, 70.295, -36.216, 2.5, -34.104, -2.07]
  Call Extruder 0.01234
  MoveL (T19429) to (107.56, 119.76, 19.9) mm, rotated rx 180 ry 0 rz -180 deg; joints [1.401, 70.295, -36.216, 2.5, -34.104, -2.07]
  Call Extruder 0.1616
  MoveL (T19430) to (103.84, 116.04, 19.9) mm, rotated rx 180 ry 0 rz -180 deg; joints [1.825, 69.173, -34.109, 3.175, -35.105, -2.598]
  Call Extruder 0.01786
  MoveL (T19431) to (103.84, 116.62, 19.9) mm, rotated rx 180 ry 0 rz -180 deg; joints [1.825, 69.173, -34.109, 3.175, -35.105, -2.598]
  Call Extruder 0.19697
  MoveL (T19432) to (108.38, 121.16, 19.9) mm, rotated rx 180 ry 0 rz -180 deg; joints [1.827, 69.002, -33.788, 3.167, -35.255, -2.587]
  Call Extruder 0.01786
  MoveL (T19433) to (107.79, 121.16, 19.9) mm, rotated rx 180 ry 0 rz -180 deg; joints [1.827, 69.002, -33.788, 3.167, -35.255, -2.587]
  Call Extruder 0.17171
  MoveL (T19434) to (103.84, 117.21, 19.9) mm, rotated rx 180 ry 0 rz -180 deg; joints [1.827, 69.002, -33.788, 3.167, -35.255, -2.587]
  Call Extruder 0.01786
  MoveL (T19435) to (103.84, 117.79, 19.9) mm, rotated rx 180 ry 0 rz -180 deg; joints [1.403, 70.115, -35.88, 2.493, -34.261, -2.06]
  Call Extruder 0.14646
  MoveL (T19436) to (107.21, 121.16, 19.9) mm, rotated rx 180 ry 0 rz -180 deg; joints [1.403, 70.115, -35.88, 2.493, -34.261, -2.06]
  Call Extruder 0.01786
  MoveL (T19437) to (106.63, 121.16, 19.9) mm, rotated rx 180 ry 0 rz -180 deg; joints [1.403, 70.115, -35.88, 2.493, -34.261, -2.06]
  Call Extruder 0.1212
  MoveL (T19438) to (103.84, 118.37, 19.9) mm, rotated rx 180 ry 0 rz -180 deg; joints [1.404, 69.938, -35.546, 2.485, -34.417, -2.051]
  Call Extruder 0.01786
  MoveL (T19439) to (103.84, 118.95, 19.9) mm, rotated rx 180 ry 0 rz -180 deg; joints [1.404, 69.938, -35.546, 2.485, -34.417, -2.051]
  Call Extruder 0.09595
  MoveL (T19440) to (106.05, 121.16, 19.9) mm, rotated rx 180 ry 0 rz -180 deg; joints [1.829, 68.832, -33.469, 3.159, -35.404, -2.576]
  Call Extruder 0.01786
  MoveL (T19441) to (105.47, 121.16, 19.9) mm, rotated rx 180 ry 0 rz -180 deg; joints [1.829, 68.832, -33.469, 3.159, -35.404, -2.576]
  Call Extruder 0.07069
  MoveL (T19442) to (103.84, 119.53, 19.9) mm, rotated rx 180 ry 0 rz -180 deg; joints [1.829, 68.832, -33.469, 3.159, -35.404, -2.576]
  Call Extruder 0.01786
  MoveL (T19443) to (103.84, 120.11, 19.9) mm, rotated rx 180 ry 0 rz -180 deg; joints [1.831, 68.728, -33.275, 3.154, -35.495, -2.569]
  Call Extruder 0.04544
  MoveL (T19444) to (104.89, 121.16, 19.9) mm, rotated rx 180 ry 0 rz -180 deg; joints [1.831, 68.728, -33.275, 3.154, -35.495, -2.569]
  Call Extruder 0.01786
  MoveL (T19445) to (104.31, 121.16, 19.9) mm, rotated rx 180 ry 0 rz -180 deg; joints [1.828, 68.714, -33.247, 3.149, -35.508, -2.564]
  Call Extruder 0.02815
  MoveL (T19446) to (103.66, 120.51, 19.9) mm, rotated rx 180 ry 0 rz -180 deg; joints [1.828, 68.714, -33.247, 3.149, -35.508, -2.564]
  Set speed (45.0 mm/s)
  Call Extruder -1.6
  MoveL (T19447) to (103.66, 120.51, 19.9) mm, rotated rx 180 ry 0 rz -180 deg; joints [1.82, 68.691, -33.204, 3.134, -35.528, -2.551]
  Set speed (120.0 mm/s)
  MoveL (T19448) to (103.66, 120.51, 19.9) mm, rotated rx 180 ry 0 rz -180 deg; joints [1.82, 68.691, -33.204, 3.134, -35.528, -2.551]
  Call Extruder -0.3262
  MoveL (T19449) to (104.31, 121.16, 19.9) mm, rotated rx 180 ry 0 rz -180 deg; joints [1.406, 69.761, -35.213, 2.478, -34.572, -2.041]
  Call Extruder -0.0538
  MoveL (T19450) to (104.46, 121.16, 19.9) mm, rotated rx 180 ry 0 rz -180 deg; joints [1.406, 69.761, -35.213, 2.478, -34.572, -2.041]
  Set speed (45.0 mm/s)
  Call Extruder -0.02
  MoveL (T19451) to (104.46, 121.16, 19.9) mm, rotated rx 180 ry 0 rz -180 deg; joints [1.406, 69.761, -35.213, 2.478, -34.572, -2.041]
  Set speed (150.0 mm/s)
  MoveL (T19452) to (104.46, 121.16, 21.9) mm, rotated rx 180 ry 0 rz -180 deg; joints [1.408, 69.586, -34.884, 2.471, -34.726, -2.032]
  MoveL (T19453) to (109.4, 105.47, 21.9) mm, rotated rx 180 ry 0 rz -180 deg; joints [1.408, 69.586, -34.884, 2.471, -34.726, -2.032]
  MoveL (T19454) to (109.4, 105.47, 20.1) mm, rotated rx 180 ry 0 rz -180 deg; joints [1.408, 69.586, -34.884, 2.471, -34.726, -2.032]
  Set speed (40.0 mm/s)
  Call Extruder 2.0
  MoveL (T19455) to (109.4, 105.47, 20.1) mm, rotated rx 180 ry 0 rz -180 deg; joints [1.79, 68.604, -33.041, 3.075, -35.602, -2.501]
  Call Extruder 0.25145
  MoveL (T19456) to (117.65, 105.47, 20.1) mm, rotated rx 180 ry 0 rz -180 deg; joints [1.79, 68.604, -33.041, 3.075, -35.602, -2.501]
  Call Extruder 0.10939
  MoveL (T19457) to (117.65, 109.06, 20.1) mm, rotated rx 180 ry 0 rz -180 deg; joints [1.79, 68.604, -33.041, 3.075, -35.602, -2.501]
  Call Extruder 0.14732
  MoveL (T19458) to (112.81, 109.06, 20.1) mm, rotated rx 180 ry 0 rz -180 deg; joints [1.759, 68.518, -32.879, 3.017, -35.676, -2.452]
  Call Extruder 0.31102
  MoveL (T19459) to (117.47, 118.15, 20.1) mm, rotated rx 180 ry 0 rz -180 deg; joints [1.759, 68.518, -32.879, 3.017, -35.676, -2.452]
  Call Extruder 0.05209
  MoveL (T19460) to (117.47, 119.86, 20.1) mm, rotated rx 180 ry 0 rz -180 deg; joints [1.409, 69.411, -34.557, 2.465, -34.879, -2.022]
  Call Extruder 0.29244
  MoveL (T19461) to (107.87, 119.86, 20.1) mm, rotated rx 180 ry 0 rz -180 deg; joints [1.411, 69.239, -34.233, 2.458, -35.03, -2.013]
  Call Extruder 0.10939
  MoveL (T19462) to (107.87, 116.27, 20.1) mm, rotated rx 180 ry 0 rz -180 deg; joints [1.411, 69.239, -34.233, 2.458, -35.03, -2.013]
  Call Extruder 0.13869
  MoveL (T19463) to (112.42, 116.27, 20.1) mm, rotated rx 180 ry 0 rz -180 deg; joints [1.728, 68.432, -32.718, 2.959, -35.75, -2.402]
  Call Extruder 0.31084
  MoveL (T19464) to (107.78, 107.18, 20.1) mm, rotated rx 180 ry 0 rz -180 deg; joints [1.728, 68.432, -32.718, 2.959, -35.75, -2.402]
  Call Extruder 0.05206
  MoveL (T19465) to (107.78, 105.47, 20.1) mm, rotated rx 180 ry 0 rz -180 deg; joints [1.698, 68.346, -32.557, 2.902, -35.824, -2.353]
  Call Extruder 0.04735
  MoveL (T19466) to (109.34, 105.47, 20.1) mm, rotated rx 180 ry 0 rz -180 deg; joints [1.698, 68.346, -32.557, 2.902, -35.824, -2.353]
  Set speed (150.0 mm/s)
  MoveL (T19467) to (109, 105.88, 20.1) mm, rotated rx 180 ry 0 rz -180 deg; joints [1.412, 69.067, -33.911, 2.451, -35.181, -2.004]
  Set speed (40.0 mm/s)
  MoveL (T19468) to (109, 105.88, 20.1) mm, rotated rx 180 ry 0 rz -180 deg; joints [1.412, 69.067, -33.911, 2.451, -35.181, -2.004]
  Call Extruder 0.25124
  MoveL (T19469) to (117.24, 105.88, 20.1) mm, rotated rx 180 ry 0 rz -180 deg; joints [1.412, 69.067, -33.911, 2.451, -35.181, -2.004]
  Call Extruder 0.08459
  MoveL (T19470) to (117.24, 108.65, 20.1) mm, rotated rx 180 ry 0 rz -180 deg; joints [1.414, 68.897, -33.591, 2.445, -35.33, -1.995]
  Call Extruder 0.1552
  MoveL (T19471) to (112.15, 108.65, 20.1) mm, rotated rx 180 ry 0 rz -180 deg; joints [1.414, 68.897, -33.591, 2.445, -35.33, -1.995]
  Call Extruder 0.32831
  MoveL (T19472) to (117.06, 118.25, 20.1) mm, rotated rx 180 ry 0 rz -180 deg; joints [1.842, 67.837, -31.6, 3.113, -36.277, -2.511]
  Call Extruder 0.0367
  MoveL (T19473) to (117.06, 119.45, 20.1) mm, rotated rx 180 ry 0 rz -180 deg; joints [1.842, 67.837, -31.6, 3.113, -36.277, -2.511]
  Call Extruder 0.26763
  MoveL (T19474) to (108.27, 119.45, 20.1) mm, rotated rx 180 ry 0 rz -180 deg; joints [1.842, 67.837, -31.6, 3.113, -36.277, -2.511]
  Call Extruder 0.08459
  MoveL (T19475) to (108.27, 116.67, 20.1) mm, rotated rx 180 ry 0 rz -180 deg; joints [1.844, 67.674, -31.296, 3.106, -36.419, -2.5]
  Call Extruder 0.14654
